Omron CX-Programmer project NewProject (CX-Programmer 9.74)

# PLC Transporte: CJ2M CPU31
I/O table (CPU CJ2M-CPU31): rack 0 slot 0 CJ1W-ID211; rack 0 slot 1 CJ1W-ID211; rack 0 slot 2 CJ1W-ID211; rack 0 slot 3 CJ1W-OD212; rack 0 slot 4 CJ1W-OD212; rack 0 slot 11 CJ2M-EIP21

## Data types
TYPE s_equip_ios : STRUCT  (* Equipamento - Entradas *)
  om : BOOL;  (* Ordem de marcha *)
  oma : BOOL;  (* Ordem de abrir *)
  omf : BOOL;  (* Ordem de fechar *)
  rm : BOOL;  (* Resposta de marcha *)
  fca : BOOL;  (* Fim de curso aberta *)
  fcf : BOOL;  (* Fim de curso fechada *)
  de : BOOL;  (* Defeito electrico *)
  pf_bmb : BOOL;  (* Pulsos de funcionamento da bomba *)
END_STRUCT END_TYPE
TYPE s_relogio : STRUCT  (* Dados de acerto e leitura de relógio *)
  pc_ano : INT;  (* Ano *)
  pc_mes : INT;  (* Mes *)
  pc_dia : INT;  (* Dia *)
  pc_dia_s : INT;  (* Dia da semana *)
  pc_hora : INT;  (* Hora *)
  pc_minuto : INT;  (* Minuto *)
  pc_segundo : INT;  (* Segundo *)
  rsv1 : INT Dimensions=[3];  (* RESERVA *)
  ano : INT;  (* Ano *)
  mes : INT;  (* Mes *)
  dia : INT;  (* Dia *)
  dia_s : INT;  (* Dia da semana *)
  hora : INT;  (* Hora *)
  minuto : INT;  (* Minuto *)
  segundo : INT;  (* Segundo *)
  rsv2 : INT Dimensions=[3];  (* RESERVA *)
END_STRUCT END_TYPE
TYPE s_caudal : STRUCT  (* Dados do caudalimetro *)
  tti : BOOL;  (* Impulso de totalização *)
  x0_1 : BOOL;  (* RESERVA *)
  x0_2 : BOOL;  (* RESERVA *)
  x0_3 : BOOL;  (* RESERVA *)
  fm : BOOL;  (* Falha de caudal *)
  rem : BOOL;  (* Totalizador local/remoto *)
  rem_ok : BOOL;  (* OK para ir buscar o valor do totalizador remoto *)
  inj_ini : BOOL;  (* Inicio da injecção *)
  x0_8 : BOOL;  (* RESERVA *)
  x0_9 : BOOL;  (* RESERVA *)
  x0_10 : BOOL;  (* RESERVA *)
  x0_11 : BOOL;  (* RESERVA *)
  x0_12 : BOOL;  (* RESERVA *)
  x0_13 : BOOL;  (* RESERVA *)
  x0_14 : BOOL;  (* RESERVA *)
  x0_15 : BOOL;  (* RESERVA *)
  prod : INT;  (* Produto *)
  rsv1 : INT Dimensions=[6];  (* RESERVA *)
  tti_x : REAL;  (* Valor do impulso *)
  tt_rem : REAL;  (* Totalizador remoto *)
  tt_rem_old : REAL;  (* Totalizador remoto antigo *)
  tt_inj : REAL;  (* Totalizador de injecção *)
  tt_p : REAL;  (* Totalizador parcial *)
  tt_g : REAL;  (* Totalizador global *)
END_STRUCT END_TYPE
TYPE s_deposito_p : STRUCT  (* Deposito de produto *)
  prod : INT;  (* Produto *)
  s_aut : BOOL;  (* Automatico *)
  mdp : BOOL;  (* Disponibilidade *)
  ndp : BOOL;  (* Não disponivel *)
  dgm : BOOL;  (* Defeito geral de maquina *)
  rst : BOOL;  (* Reset *)
  on : BOOL;  (* Deposito ligado *)
  oms_red : BOOL;  (* Lampada FLASH vermelho *)
  oms_green : BOOL;  (* Lampada FLASH verde *)
  rsv1 : INT Dimensions=[8];  (* Reserva *)
END_STRUCT END_TYPE
TYPE s_equip_bits : STRUCT  (* Equipamento - Bits auxiliares *)
  s_aut : BOOL;  (* Automatico *)
  mdp : BOOL;  (* Disponibilidade *)
  ndp : BOOL;  (* Não disponivel *)
  dgm : BOOL;  (* Defeito geral de maquina *)
  rst : BOOL;  (* Reset *)
  cfa : BOOL;  (* Condição de funcionamento automatico *)
  cfm : BOOL;  (* Condição de funcionamento manual *)
  cfaa : BOOL;  (* Condição de funcionamento automatico abrir *)
  cfaf : BOOL;  (* Condição de funcionamento automatico fechar *)
  cfma : BOOL;  (* Condição de funcionamento manual abrir *)
  cfmf : BOOL;  (* Condição de funcionamento manual fechar *)
  st_hmi : BOOL;  (* Arranque HMI *)
  sp_hmi : BOOL;  (* Paragem HMI *)
  p_hmi : BOOL;  (* Pausa HMI *)
END_STRUCT END_TYPE
TYPE s_equip_defs : STRUCT  (* Equipamentos - Defeitos *)
  fm : BOOL;  (* Falha de marcha *)
  fma : BOOL;  (* Falha de manobra abrir *)
  fmf : BOOL;  (* Falha de manobra fechar *)
  de : BOOL;  (* Defeito electrico *)
  dv : BOOL;  (* Deposito vazio *)
END_STRUCT END_TYPE
TYPE s_equip : STRUCT  (* Equipamento *)
  ios : s_equip_ios;  (* Entradas *)
  bits : s_equip_bits;  (* Bits *)
  defs : s_equip_defs;  (* Defeitos *)
  es : INT;  (* Estado *)
  tm_b : INT;  (* Tempo entre bombagens *)
  rsv1 : INT Dimensions=[5];  (* Reserva *)
END_STRUCT END_TYPE

## Global symbols (name address type ; comment)
Actv_M E0_25101 INT
H0.00 BOOL  ; CDTs Visible
Auto_Transport FIFO
Auto_Trspt_EN E0_25100.06 BOOL
Last_Rqst E0_25102 INT
Priority_Array E0_25000 INT[100]
Tapete1 fb_eq_motor
Tapete2 fb_eq_motor
Tapete3 fb_eq_motor
Tapete4 fb_eq_motor
Trspt_Array_Full E0_25100.07 BOOL
Trspt_Free E0_25100.14 BOOL
comm_M1_Rqst E0_25100.00 BOOL  ; From MES1
comm_M2_Rqst E0_25100.01 BOOL  ; From MES1
comm_M3_Rqst E0_25100.02 BOOL  ; From MES1
comm_M4_Rqst E0_25100.03 BOOL  ; From MES1
comm_M5_Rqst E0_25100.04 BOOL  ; From MES2
comm_M6_Rqst E0_25100.05 BOOL  ; From MES2
fb_eq_vc_M1 fb_eq_valvula
fb_eq_vc_M2 fb_eq_valvula
fb_eq_vc_M3 fb_eq_valvula
fb_eq_vc_M4 fb_eq_valvula
fb_eq_vc_M5 fb_eq_valvula
fb_eq_vc_M6 fb_eq_valvula
fb_eq_vd_M1 fb_eq_valvula
fb_eq_vd_M2 fb_eq_valvula
fb_eq_vd_M3 fb_eq_valvula
fb_eq_vd_M4 fb_eq_valvula
fb_eq_vd_M5 fb_eq_valvula
fb_eq_vd_M6 fb_eq_valvula

## Program Transporte (cyclic task 0)
Local symbols
Alarme_naa_t1 D0.01 BOOL
Alim_M1 W1.00 BOOL
Alim_M2 W1.01 BOOL
Alim_M3 W1.02 BOOL
Alim_M4 W1.03 BOOL
Alim_M5 W1.04 BOOL
Alim_M6 W1.05 BOOL
Carga_M1 D10050.05 BOOL  ; Ordem de alimentação da Máquina 1
Carga_M2 D10100.05 BOOL  ; Ordem de alimentação da Máquina 2
Carga_M3 D10150.05 BOOL  ; Ordem de alimentação da Máquina 3
Carga_M4 D10200.05 BOOL  ; Ordem de alimentação da Máquina 4
Carga_M5 D10250.05 BOOL  ; Ordem de alimentação da Máquina 5
Carga_M6 D10300.05 BOOL  ; Ordem de alimentação da Máquina 6
Encravamento_t2 W0.00 BOOL
M1_TrpRqst_Holder W2.02 BOOL
M2_TrpRqstHolder BOOL
M2_TrpRqst_Holder W2.00 BOOL
M3_TrpRqst_Holder W2.01 BOOL
M4_TrpRqst_Holder W2.03 BOOL
M5_TrpRqst_Holder W2.05 BOOL
M6_TrpRqst_Holder W2.04 BOOL
Tapete1 D10 STRUCT s_equip
Tapete2 D20 STRUCT s_equip
Tapete3 D30 STRUCT s_equip
Tapete4 D40 STRUCT s_equip
Transporte_M1 E0_25100.08 BOOL  ; Ordem de alimentação do Silo da Máquina 1
Transporte_M2 E0_25100.09 BOOL  ; Ordem de alimentação do Silo da Máquina 2
Transporte_M3 E0_25100.10 BOOL  ; Ordem de alimentação do Silo da Máquina 3
Transporte_M4 E0_25100.11 BOOL  ; Ordem de alimentação do Silo da Máquina 4
Transporte_M5 E0_25100.12 BOOL  ; Ordem de alimentação do Silo da Máquina 5
Transporte_M6 E0_25100.13 BOOL  ; Ordem de alimentação do Silo da Máquina 6
al_na_m1 D2.01 BOOL  ; Nivel alto estabilizado maquina 1
al_na_m2 D2.02 BOOL  ; Nivel alto estabilizado maquina 2
al_na_m3 D2.03 BOOL  ; Nivel alto estabilizado maquina 3
al_na_m4 D2.04 BOOL  ; Nivel alto estabilizado maquina 4
al_na_m5 D2.05 BOOL  ; Nivel alto estabilizado maquina 5
al_na_m6 D2.06 BOOL  ; Nivel alto estabilizado maquina 6
al_nb_m1 D1.01 BOOL  ; Nivel baixo estabilizado maquina 1
al_nb_m2 D1.02 BOOL  ; Nivel baixo estabilizado maquina 2
al_nb_m3 D1.03 BOOL  ; Nivel baixo estabilizado maquina 3
al_nb_m4 D1.04 BOOL  ; Nivel baixo estabilizado maquina 4
al_nb_m5 D1.05 BOOL  ; Nivel baixo estabilizado maquina 5
al_nb_m6 D1.06 BOOL  ; Nivel baixo estabilizado maquina 6
cmd_rst_vc_M1 D10050.03 BOOL  ; Comando de reset da Razeira da Máquina 1
cmd_rst_vc_M2 D10100.03 BOOL  ; Comando de reset da Razeira da Máquina 2
cmd_rst_vc_M3 D10150.03 BOOL  ; Comando de reset da Razeira da Máquina 3
cmd_rst_vc_M4 D10200.03 BOOL  ; Comando de reset da Razeira da Máquina 4
cmd_rst_vc_M5 D10250.03 BOOL  ; Comando de reset da Razeira da Máquina 5
cmd_rst_vc_M6 D10300.03 BOOL  ; Comando de reset da Razeira da Máquina 6
cmd_tp3_M1 D10050.06 BOOL  ; Ordem de marcha Tapete 3 a partir da Máquina 1
cmd_tp3_M2 D10100.06 BOOL  ; Ordem de marcha Tapete 3 a partir da Máquina 2
cmd_tp3_M3 D10150.06 BOOL  ; Ordem de marcha Tapete 3 a partir da Máquina 3
cmd_tp3_M4 D10200.06 BOOL  ; Ordem de marcha Tapete 3 a partir da Máquina 4
cmd_tp3_M5 D10250.06 BOOL  ; Ordem de marcha Tapete 3 a partir da Máquina 5
cmd_tp3_M6 D10300.06 BOOL  ; Ordem de marcha Tapete 3 a partir da Máquina 6
cmd_tp4_M1 D10050.07 BOOL  ; Ordem de marcha Tapete 4 a partir da Máquina 1
cmd_tp4_M2 D10100.07 BOOL  ; Ordem de marcha Tapete 4 a partir da Máquina 2
cmd_tp4_M3 D10150.07 BOOL  ; Ordem de marcha Tapete 4 a partir da Máquina 3
cmd_tp4_M4 D10200.07 BOOL  ; Ordem de marcha Tapete 4 a partir da Máquina 4
cmd_tp4_M5 D10250.07 BOOL  ; Ordem de marcha Tapete 4 a partir da Máquina 5
cmd_tp4_M6 D10300.07 BOOL  ; Ordem de marcha Tapete 4 a partir da Máquina 6
de_t1 1.00 BOOL  ; Disparo termico no tapete 1
de_t2 1.01 BOOL  ; Disparo termico no tapete 2
de_t3 1.02 BOOL  ; Disparo termico no tapete 3
de_t4 1.03 BOOL  ; Disparo termico no tapete 4
disp_transporte D0.03 BOOL
fca_vd_m1 2.00 BOOL  ; Valvula desviadora aberta - maquina 1
fca_vd_m2 2.02 BOOL  ; Valvula desviadora aberta - maquina 2
fca_vd_m3 2.04 BOOL  ; Valvula desviadora aberta - maquina 3
fca_vd_m4 2.06 BOOL  ; Valvula desviadora aberta - maquina 4
fca_vd_m5 2.08 BOOL  ; Valvula desviadora aberta - maquina 5
fca_vd_m6 2.10 BOOL  ; Valvula desviadora aberta - maquina 6
fcf_vc_m1 1.04 BOOL  ; Razeira de carga fechada - maquina 1
fcf_vc_m2 1.05 BOOL  ; Razeira de carga fechada - maquina 2
fcf_vc_m3 1.06 BOOL  ; Razeira de carga fechada - maquina 3
fcf_vc_m4 1.07 BOOL  ; Razeira de carga fechada - maquina 4
fcf_vc_m5 1.08 BOOL  ; Razeira de carga fechada - maquina 5
fcf_vc_m6 1.09 BOOL  ; Razeira de carga fechada - maquina 6
fcf_vd_m1 2.01 BOOL  ; Valvula desviadora fechada - maquina 1
fcf_vd_m2 2.03 BOOL  ; Valvula desviadora fechada - maquina 2
fcf_vd_m3 2.05 BOOL  ; Valvula desviadora fechada - maquina 3
fcf_vd_m4 2.07 BOOL  ; Valvula desviadora fechada - maquina 4
fcf_vd_m5 2.09 BOOL  ; Valvula desviadora fechada - maquina 5
fcf_vd_m6 2.11 BOOL  ; Valvula desviadora fechada - maquina 6
msb_1 BOOL
na_m1 0.02 BOOL  ; Nivel alto na moega de carga maquina 1
na_m2 0.04 BOOL  ; Nivel alto na moega de carga maquina 2
na_m3 0.06 BOOL  ; Nivel alto na moega de carga maquina 3
na_m4 0.08 BOOL  ; Nivel alto na moega de carga maquina 4
na_m5 0.10 BOOL  ; Nivel alto na moega de carga maquina 5
na_m6 0.12 BOOL  ; Nivel alto na moega de carga maquina 6
naa_t1 0.14 BOOL  ; Nivel muito alto no tapete 1
naa_t1_tp D0.00 BOOL
nb_m1 0.03 BOOL  ; Nivel baixo na moega de carga maquina 1
nb_m2 0.05 BOOL  ; Nivel baixo na moega de carga maquina 2
nb_m3 0.07 BOOL  ; Nivel baixo na moega de carga maquina 3
nb_m4 0.09 BOOL  ; Nivel baixo na moega de carga maquina 4
nb_m5 0.11 BOOL  ; Nivel baixo na moega de carga maquina 5
nb_m6 0.13 BOOL  ; Nivel baixo na moega de carga maquina 6
om_t1 3.00 BOOL  ; Ordem de marcha tapete 1
om_t2 3.01 BOOL  ; Ordem de marcha tapete 2
om_t3 3.02 BOOL  ; Ordem de marcha tapete 3
om_t4 3.03 BOOL  ; Ordem de marcha tapete 4
oma_vc_m1 3.04 BOOL  ; Abrir razeira de carga - maquina 1
oma_vc_m2 3.06 BOOL  ; Abrir razeira de carga - maquina 2
oma_vc_m3 3.08 BOOL  ; Abrir razeira de carga - maquina 3
oma_vc_m4 3.10 BOOL  ; Abrir razeira de carga - maquina 4
oma_vc_m5 3.12 BOOL  ; Abrir razeira de carga - maquina 5
oma_vc_m6 3.14 BOOL  ; Abrir razeira de carga - maquina 6
oma_vd_m1 4.01 BOOL  ; Abrir valvula desviadora - maquina 1
oma_vd_m2 4.03 BOOL  ; Abrir valvula desviadora - maquina 2
oma_vd_m3 4.05 BOOL  ; Abrir valvula desviadora - maquina 3
oma_vd_m4 4.07 BOOL  ; Abrir valvula desviadora - maquina 4
oma_vd_m5 4.09 BOOL  ; Abrir valvula desviadora - maquina 5
oma_vd_m6 4.11 BOOL  ; Abrir valvula desviadora - maquina 6
omf_vc_m1 3.05 BOOL  ; Fechar razeira de carga - maquina 1
omf_vc_m2 3.07 BOOL  ; Fechar razeira de carga - maquina 2
omf_vc_m3 3.09 BOOL  ; Fechar razeira de carga - maquina 3
omf_vc_m4 3.11 BOOL  ; Fechar razeira de carga - maquina 4
omf_vc_m5 3.13 BOOL  ; Fechar razeira de carga - maquina 5
omf_vc_m6 3.15 BOOL  ; Fechar razeira de carga - maquina 6
omf_vd_m1 4.00 BOOL  ; Fechar valvula desviadora - maquina 1
omf_vd_m2 4.02 BOOL  ; Fechar valvula desviadora - maquina 2
omf_vd_m3 4.04 BOOL  ; Fechar valvula desviadora - maquina 3
omf_vd_m4 4.06 BOOL  ; Fechar valvula desviadora - maquina 4
omf_vd_m5 4.08 BOOL  ; Fechar valvula desviadora - maquina 5
omf_vd_m6 4.10 BOOL  ; Fechar valvula desviadora - maquina 6
pe_transporte 0.00 BOOL  ; Botoneira de Emergência
rem_transporte 0.01 BOOL  ; Automatico
rm_t1 1.10 BOOL  ; Resposta de marcha tapete 1
rm_t2 1.11 BOOL  ; Resposta de marcha tapete 2
rm_t3 1.12 BOOL  ; Resposta de marcha tapete 3
rm_t4 1.13 BOOL  ; Resposta de marcha tapete 4
rm_transporte D0.05 BOOL
so_1alim D0.02 BOOL
stop_transporte D0.04 BOOL
vc_M1 D100 STRUCT s_equip
vc_M2 D110 STRUCT s_equip
vc_M3 D120 STRUCT s_equip
vc_M4 D130 STRUCT s_equip
vc_M5 D140 STRUCT s_equip
vc_M6 D150 STRUCT s_equip
vd_M1 D200 STRUCT s_equip
vd_M2 D210 STRUCT s_equip
vd_M3 D220 STRUCT s_equip
vd_M4 D230 STRUCT s_equip
vd_M5 D240 STRUCT s_equip
vd_M6 D250 STRUCT s_equip

### Section Valvulas

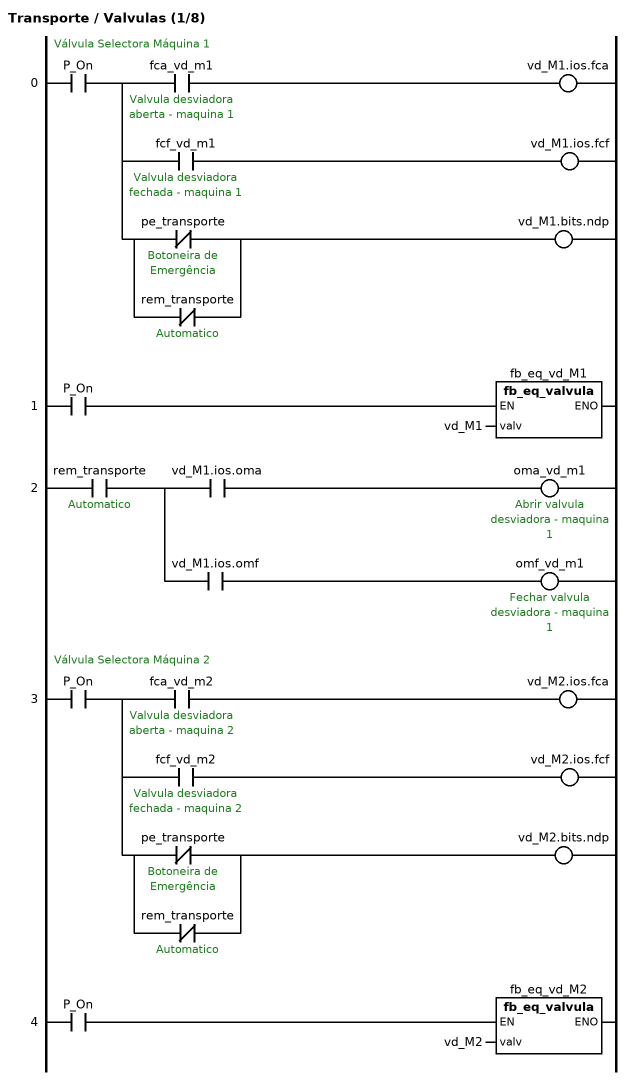
; rung 0: Válvula Selectora Máquina 1
LD P_On
OUT TR0
AND fca_vd_m1  ; Valvula desviadora aberta - maquina 1
OUT vd_M1.ios.fca
LD TR0
AND fcf_vd_m1  ; Valvula desviadora fechada - maquina 1
OUT vd_M1.ios.fcf
LD TR0
LDNOT pe_transporte  ; Botoneira de Emergência
ORNOT rem_transporte  ; Automatico
ANDLD
OUT vd_M1.bits.ndp
; rung 1
LD P_On
CALL fb_eq_vd_M1 : fb_eq_valvula (valv := vd_M1)
; rung 2
LD rem_transporte  ; Automatico
OUT TR0
AND vd_M1.ios.oma
OUT oma_vd_m1  ; Abrir valvula desviadora - maquina 1
LD TR0
AND vd_M1.ios.omf
OUT omf_vd_m1  ; Fechar valvula desviadora - maquina 1
; rung 3: Válvula Selectora Máquina 2
LD P_On
OUT TR0
AND fca_vd_m2  ; Valvula desviadora aberta - maquina 2
OUT vd_M2.ios.fca
LD TR0
AND fcf_vd_m2  ; Valvula desviadora fechada - maquina 2
OUT vd_M2.ios.fcf
LD TR0
LDNOT pe_transporte  ; Botoneira de Emergência
ORNOT rem_transporte  ; Automatico
ANDLD
OUT vd_M2.bits.ndp
; rung 4
LD P_On
CALL fb_eq_vd_M2 : fb_eq_valvula (valv := vd_M2)

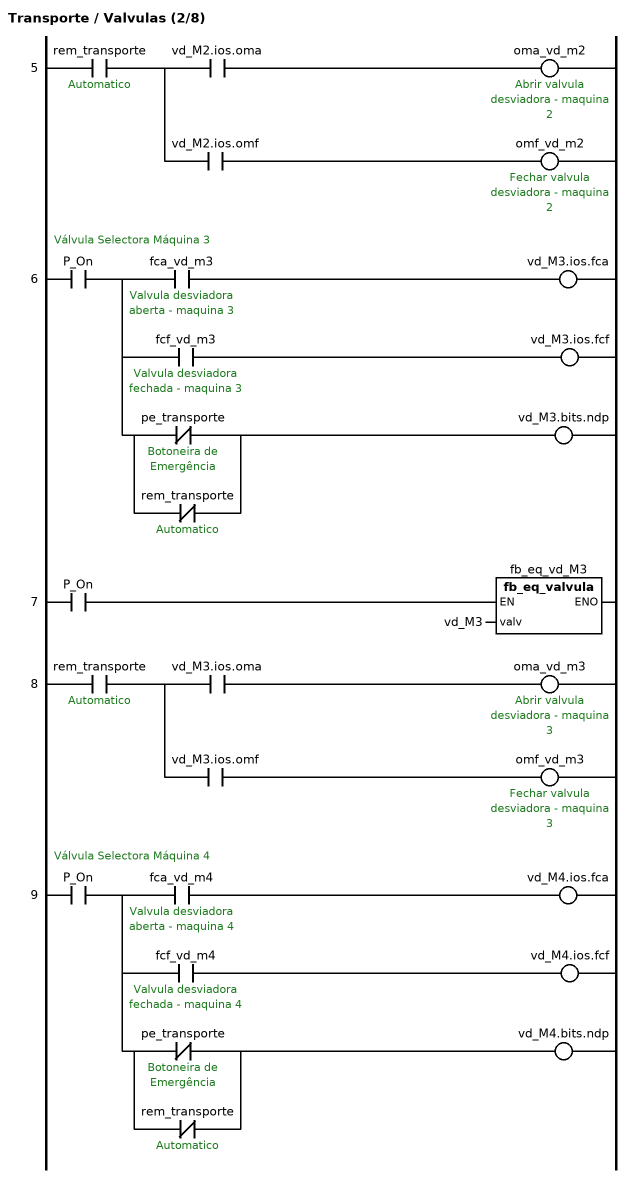
; rung 5
LD rem_transporte  ; Automatico
OUT TR0
AND vd_M2.ios.oma
OUT oma_vd_m2  ; Abrir valvula desviadora - maquina 2
LD TR0
AND vd_M2.ios.omf
OUT omf_vd_m2  ; Fechar valvula desviadora - maquina 2
; rung 6: Válvula Selectora Máquina 3
LD P_On
OUT TR0
AND fca_vd_m3  ; Valvula desviadora aberta - maquina 3
OUT vd_M3.ios.fca
LD TR0
AND fcf_vd_m3  ; Valvula desviadora fechada - maquina 3
OUT vd_M3.ios.fcf
LD TR0
LDNOT pe_transporte  ; Botoneira de Emergência
ORNOT rem_transporte  ; Automatico
ANDLD
OUT vd_M3.bits.ndp
; rung 7
LD P_On
CALL fb_eq_vd_M3 : fb_eq_valvula (valv := vd_M3)
; rung 8
LD rem_transporte  ; Automatico
OUT TR0
AND vd_M3.ios.oma
OUT oma_vd_m3  ; Abrir valvula desviadora - maquina 3
LD TR0
AND vd_M3.ios.omf
OUT omf_vd_m3  ; Fechar valvula desviadora - maquina 3
; rung 9: Válvula Selectora Máquina 4
LD P_On
OUT TR0
AND fca_vd_m4  ; Valvula desviadora aberta - maquina 4
OUT vd_M4.ios.fca
LD TR0
AND fcf_vd_m4  ; Valvula desviadora fechada - maquina 4
OUT vd_M4.ios.fcf
LD TR0
LDNOT pe_transporte  ; Botoneira de Emergência
ORNOT rem_transporte  ; Automatico
ANDLD
OUT vd_M4.bits.ndp

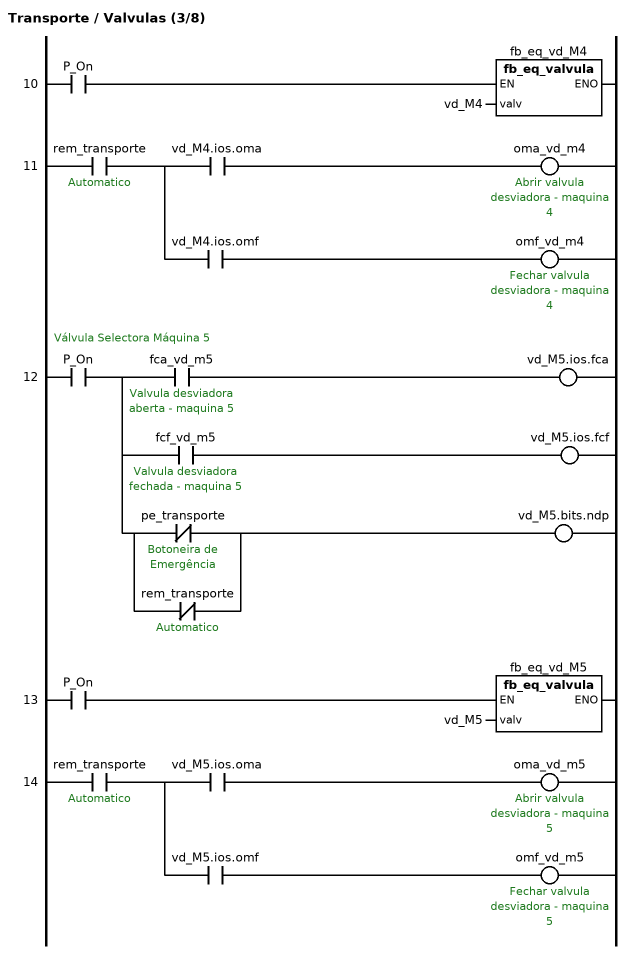
; rung 10
LD P_On
CALL fb_eq_vd_M4 : fb_eq_valvula (valv := vd_M4)
; rung 11
LD rem_transporte  ; Automatico
OUT TR0
AND vd_M4.ios.oma
OUT oma_vd_m4  ; Abrir valvula desviadora - maquina 4
LD TR0
AND vd_M4.ios.omf
OUT omf_vd_m4  ; Fechar valvula desviadora - maquina 4
; rung 12: Válvula Selectora Máquina 5
LD P_On
OUT TR0
AND fca_vd_m5  ; Valvula desviadora aberta - maquina 5
OUT vd_M5.ios.fca
LD TR0
AND fcf_vd_m5  ; Valvula desviadora fechada - maquina 5
OUT vd_M5.ios.fcf
LD TR0
LDNOT pe_transporte  ; Botoneira de Emergência
ORNOT rem_transporte  ; Automatico
ANDLD
OUT vd_M5.bits.ndp
; rung 13
LD P_On
CALL fb_eq_vd_M5 : fb_eq_valvula (valv := vd_M5)
; rung 14
LD rem_transporte  ; Automatico
OUT TR0
AND vd_M5.ios.oma
OUT oma_vd_m5  ; Abrir valvula desviadora - maquina 5
LD TR0
AND vd_M5.ios.omf
OUT omf_vd_m5  ; Fechar valvula desviadora - maquina 5

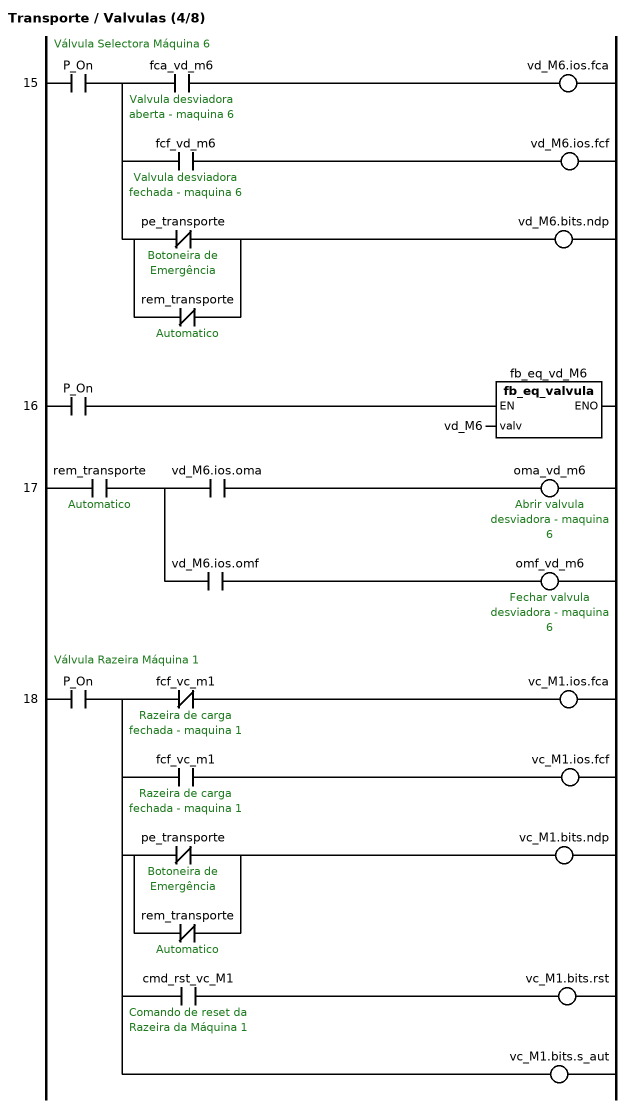
; rung 15: Válvula Selectora Máquina 6
LD P_On
OUT TR0
AND fca_vd_m6  ; Valvula desviadora aberta - maquina 6
OUT vd_M6.ios.fca
LD TR0
AND fcf_vd_m6  ; Valvula desviadora fechada - maquina 6
OUT vd_M6.ios.fcf
LD TR0
LDNOT pe_transporte  ; Botoneira de Emergência
ORNOT rem_transporte  ; Automatico
ANDLD
OUT vd_M6.bits.ndp
; rung 16
LD P_On
CALL fb_eq_vd_M6 : fb_eq_valvula (valv := vd_M6)
; rung 17
LD rem_transporte  ; Automatico
OUT TR0
AND vd_M6.ios.oma
OUT oma_vd_m6  ; Abrir valvula desviadora - maquina 6
LD TR0
AND vd_M6.ios.omf
OUT omf_vd_m6  ; Fechar valvula desviadora - maquina 6
; rung 18: Válvula Razeira Máquina 1
LD P_On
OUT TR0
ANDNOT fcf_vc_m1  ; Razeira de carga fechada - maquina 1
OUT vc_M1.ios.fca
LD TR0
AND fcf_vc_m1  ; Razeira de carga fechada - maquina 1
OUT vc_M1.ios.fcf
LD TR0
LDNOT pe_transporte  ; Botoneira de Emergência
ORNOT rem_transporte  ; Automatico
ANDLD
OUT vc_M1.bits.ndp
LD TR0
AND cmd_rst_vc_M1  ; Comando de reset da Razeira da Máquina 1
OUT vc_M1.bits.rst
LD TR0
OUT vc_M1.bits.s_aut

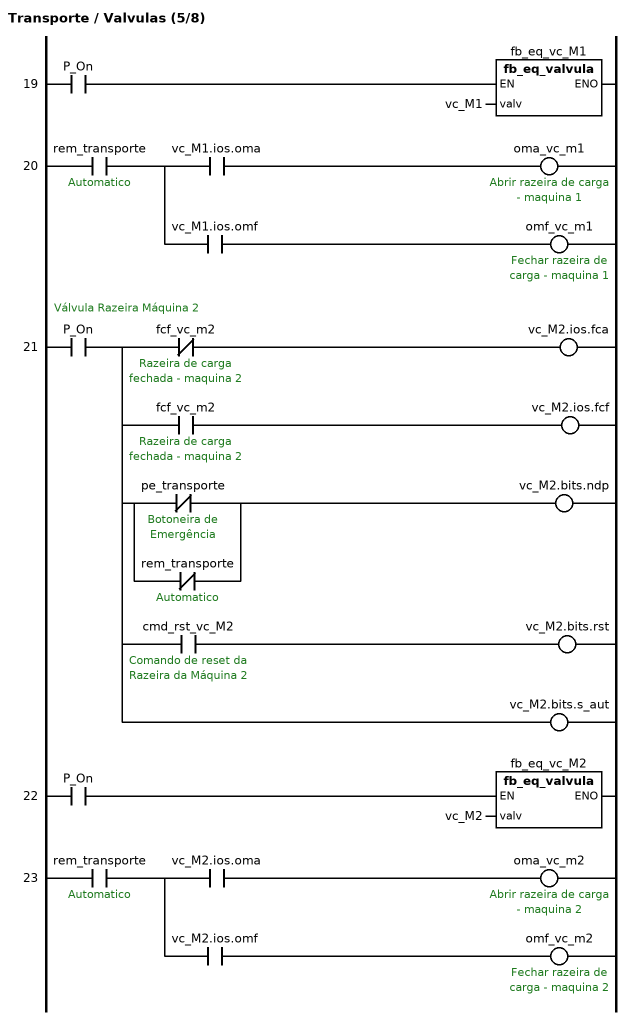
; rung 19
LD P_On
CALL fb_eq_vc_M1 : fb_eq_valvula (valv := vc_M1)
; rung 20
LD rem_transporte  ; Automatico
OUT TR0
AND vc_M1.ios.oma
OUT oma_vc_m1  ; Abrir razeira de carga - maquina 1
LD TR0
AND vc_M1.ios.omf
OUT omf_vc_m1  ; Fechar razeira de carga - maquina 1
; rung 21: Válvula Razeira Máquina 2
LD P_On
OUT TR0
ANDNOT fcf_vc_m2  ; Razeira de carga fechada - maquina 2
OUT vc_M2.ios.fca
LD TR0
AND fcf_vc_m2  ; Razeira de carga fechada - maquina 2
OUT vc_M2.ios.fcf
LD TR0
LDNOT pe_transporte  ; Botoneira de Emergência
ORNOT rem_transporte  ; Automatico
ANDLD
OUT vc_M2.bits.ndp
LD TR0
AND cmd_rst_vc_M2  ; Comando de reset da Razeira da Máquina 2
OUT vc_M2.bits.rst
LD TR0
OUT vc_M2.bits.s_aut
; rung 22
LD P_On
CALL fb_eq_vc_M2 : fb_eq_valvula (valv := vc_M2)
; rung 23
LD rem_transporte  ; Automatico
OUT TR0
AND vc_M2.ios.oma
OUT oma_vc_m2  ; Abrir razeira de carga - maquina 2
LD TR0
AND vc_M2.ios.omf
OUT omf_vc_m2  ; Fechar razeira de carga - maquina 2

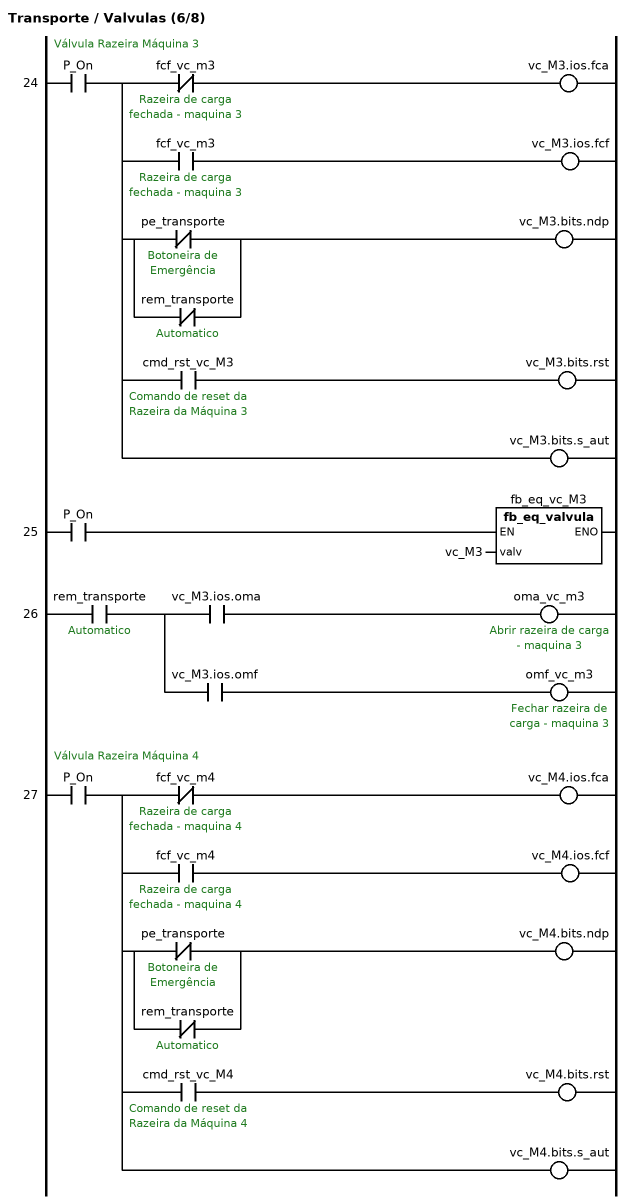
; rung 24: Válvula Razeira Máquina 3
LD P_On
OUT TR0
ANDNOT fcf_vc_m3  ; Razeira de carga fechada - maquina 3
OUT vc_M3.ios.fca
LD TR0
AND fcf_vc_m3  ; Razeira de carga fechada - maquina 3
OUT vc_M3.ios.fcf
LD TR0
LDNOT pe_transporte  ; Botoneira de Emergência
ORNOT rem_transporte  ; Automatico
ANDLD
OUT vc_M3.bits.ndp
LD TR0
AND cmd_rst_vc_M3  ; Comando de reset da Razeira da Máquina 3
OUT vc_M3.bits.rst
LD TR0
OUT vc_M3.bits.s_aut
; rung 25
LD P_On
CALL fb_eq_vc_M3 : fb_eq_valvula (valv := vc_M3)
; rung 26
LD rem_transporte  ; Automatico
OUT TR0
AND vc_M3.ios.oma
OUT oma_vc_m3  ; Abrir razeira de carga - maquina 3
LD TR0
AND vc_M3.ios.omf
OUT omf_vc_m3  ; Fechar razeira de carga - maquina 3
; rung 27: Válvula Razeira Máquina 4
LD P_On
OUT TR0
ANDNOT fcf_vc_m4  ; Razeira de carga fechada - maquina 4
OUT vc_M4.ios.fca
LD TR0
AND fcf_vc_m4  ; Razeira de carga fechada - maquina 4
OUT vc_M4.ios.fcf
LD TR0
LDNOT pe_transporte  ; Botoneira de Emergência
ORNOT rem_transporte  ; Automatico
ANDLD
OUT vc_M4.bits.ndp
LD TR0
AND cmd_rst_vc_M4  ; Comando de reset da Razeira da Máquina 4
OUT vc_M4.bits.rst
LD TR0
OUT vc_M4.bits.s_aut

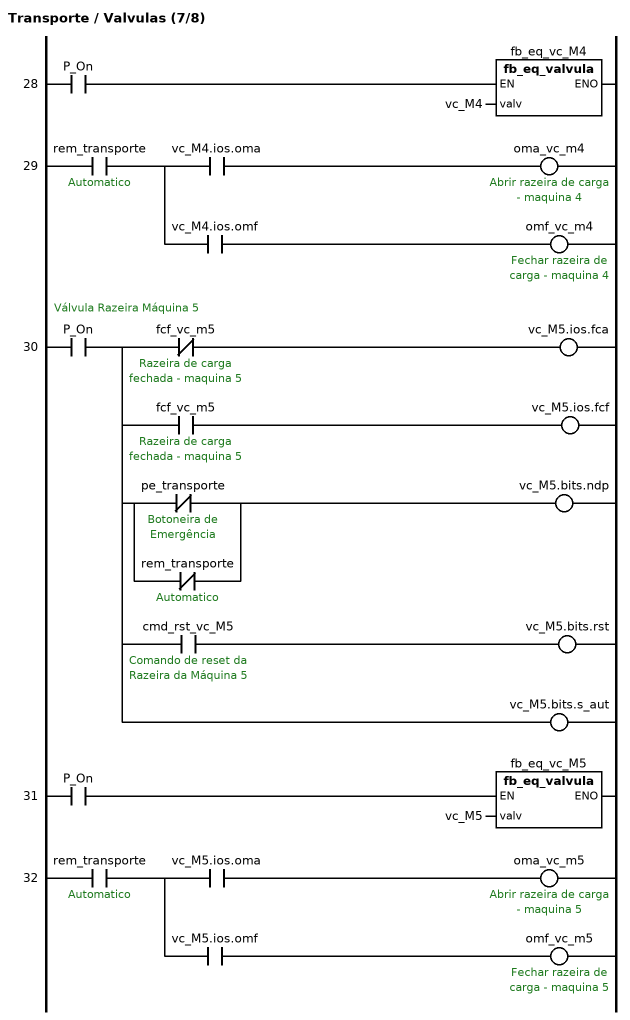
; rung 28
LD P_On
CALL fb_eq_vc_M4 : fb_eq_valvula (valv := vc_M4)
; rung 29
LD rem_transporte  ; Automatico
OUT TR0
AND vc_M4.ios.oma
OUT oma_vc_m4  ; Abrir razeira de carga - maquina 4
LD TR0
AND vc_M4.ios.omf
OUT omf_vc_m4  ; Fechar razeira de carga - maquina 4
; rung 30: Válvula Razeira Máquina 5
LD P_On
OUT TR0
ANDNOT fcf_vc_m5  ; Razeira de carga fechada - maquina 5
OUT vc_M5.ios.fca
LD TR0
AND fcf_vc_m5  ; Razeira de carga fechada - maquina 5
OUT vc_M5.ios.fcf
LD TR0
LDNOT pe_transporte  ; Botoneira de Emergência
ORNOT rem_transporte  ; Automatico
ANDLD
OUT vc_M5.bits.ndp
LD TR0
AND cmd_rst_vc_M5  ; Comando de reset da Razeira da Máquina 5
OUT vc_M5.bits.rst
LD TR0
OUT vc_M5.bits.s_aut
; rung 31
LD P_On
CALL fb_eq_vc_M5 : fb_eq_valvula (valv := vc_M5)
; rung 32
LD rem_transporte  ; Automatico
OUT TR0
AND vc_M5.ios.oma
OUT oma_vc_m5  ; Abrir razeira de carga - maquina 5
LD TR0
AND vc_M5.ios.omf
OUT omf_vc_m5  ; Fechar razeira de carga - maquina 5

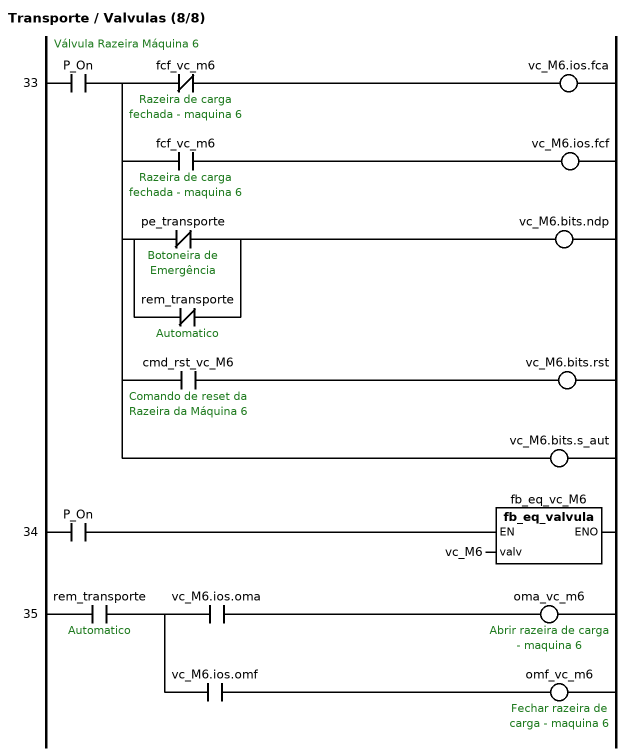
; rung 33: Válvula Razeira Máquina 6
LD P_On
OUT TR0
ANDNOT fcf_vc_m6  ; Razeira de carga fechada - maquina 6
OUT vc_M6.ios.fca
LD TR0
AND fcf_vc_m6  ; Razeira de carga fechada - maquina 6
OUT vc_M6.ios.fcf
LD TR0
LDNOT pe_transporte  ; Botoneira de Emergência
ORNOT rem_transporte  ; Automatico
ANDLD
OUT vc_M6.bits.ndp
LD TR0
AND cmd_rst_vc_M6  ; Comando de reset da Razeira da Máquina 6
OUT vc_M6.bits.rst
LD TR0
OUT vc_M6.bits.s_aut
; rung 34
LD P_On
CALL fb_eq_vc_M6 : fb_eq_valvula (valv := vc_M6)
; rung 35
LD rem_transporte  ; Automatico
OUT TR0
AND vc_M6.ios.oma
OUT oma_vc_m6  ; Abrir razeira de carga - maquina 6
LD TR0
AND vc_M6.ios.omf
OUT omf_vc_m6  ; Fechar razeira de carga - maquina 6

### Section Tapetes

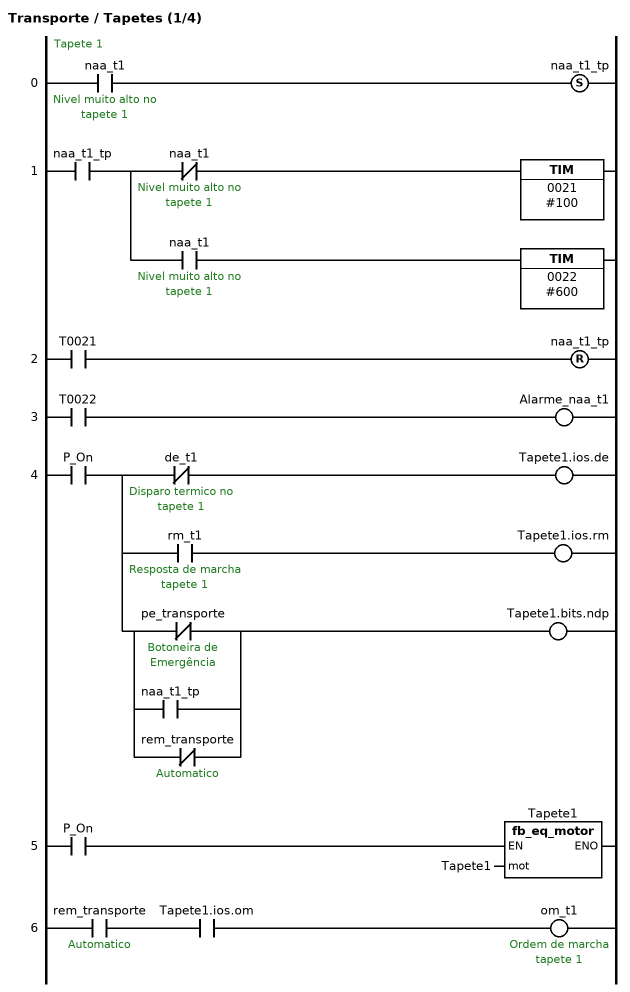
; rung 0: Tapete 1
LD naa_t1  ; Nivel muito alto no tapete 1
SET naa_t1_tp
; rung 1
LD naa_t1_tp
OUT TR0
ANDNOT naa_t1  ; Nivel muito alto no tapete 1
TIM 0021 #100
LD TR0
AND naa_t1  ; Nivel muito alto no tapete 1
TIM 0022 #600
; rung 2
LD T0021
RSET naa_t1_tp
; rung 3
LD T0022
OUT Alarme_naa_t1
; rung 4
LD P_On
OUT TR0
ANDNOT de_t1  ; Disparo termico no tapete 1
OUT Tapete1.ios.de
LD TR0
AND rm_t1  ; Resposta de marcha tapete 1
OUT Tapete1.ios.rm
LD TR0
LDNOT pe_transporte  ; Botoneira de Emergência
OR naa_t1_tp
ORNOT rem_transporte  ; Automatico
ANDLD
OUT Tapete1.bits.ndp
; rung 5
LD P_On
CALL Tapete1 : fb_eq_motor (mot := Tapete1)
; rung 6
LD rem_transporte  ; Automatico
AND Tapete1.ios.om
OUT om_t1  ; Ordem de marcha tapete 1

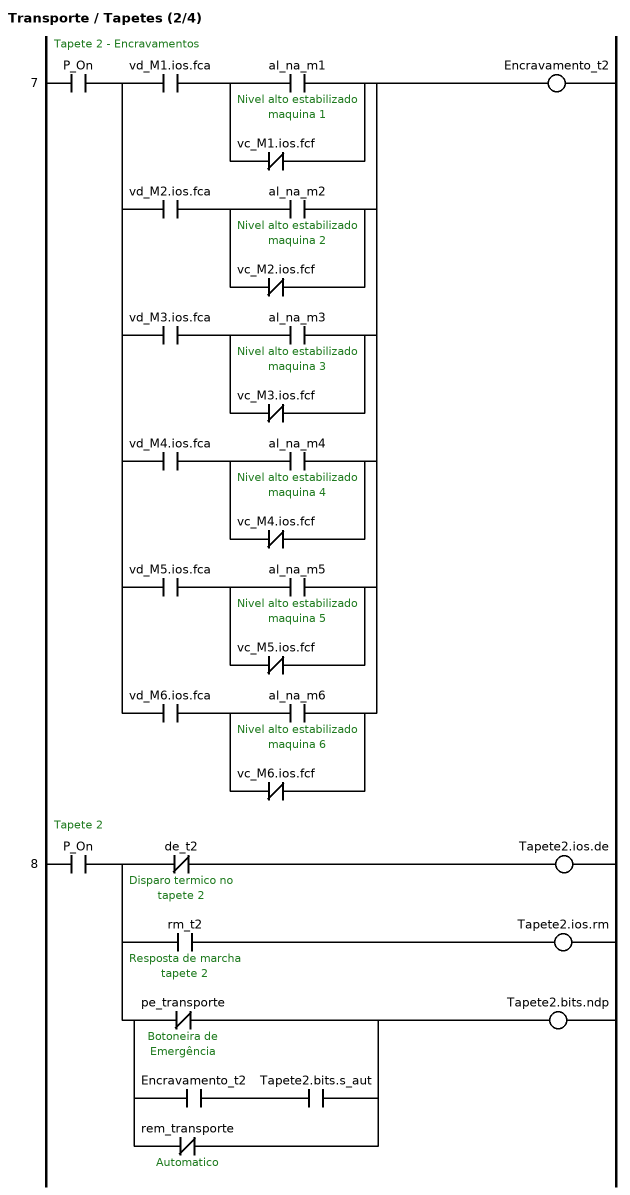
; rung 7: Tapete 2 - Encravamentos
LD P_On
LD vd_M1.ios.fca
LD al_na_m1  ; Nivel alto estabilizado maquina 1
ORNOT vc_M1.ios.fcf
ANDLD
LD vd_M2.ios.fca
LD al_na_m2  ; Nivel alto estabilizado maquina 2
ORNOT vc_M2.ios.fcf
ANDLD
ORLD
LD vd_M3.ios.fca
LD al_na_m3  ; Nivel alto estabilizado maquina 3
ORNOT vc_M3.ios.fcf
ANDLD
ORLD
LD vd_M4.ios.fca
LD al_na_m4  ; Nivel alto estabilizado maquina 4
ORNOT vc_M4.ios.fcf
ANDLD
ORLD
LD vd_M5.ios.fca
LD al_na_m5  ; Nivel alto estabilizado maquina 5
ORNOT vc_M5.ios.fcf
ANDLD
ORLD
LD vd_M6.ios.fca
LD al_na_m6  ; Nivel alto estabilizado maquina 6
ORNOT vc_M6.ios.fcf
ANDLD
ORLD
ANDLD
OUT Encravamento_t2
; rung 8: Tapete 2
LD P_On
OUT TR0
ANDNOT de_t2  ; Disparo termico no tapete 2
OUT Tapete2.ios.de
LD TR0
AND rm_t2  ; Resposta de marcha tapete 2
OUT Tapete2.ios.rm
LD TR0
LDNOT pe_transporte  ; Botoneira de Emergência
LD Encravamento_t2
AND Tapete2.bits.s_aut
ORLD
ORNOT rem_transporte  ; Automatico
ANDLD
OUT Tapete2.bits.ndp

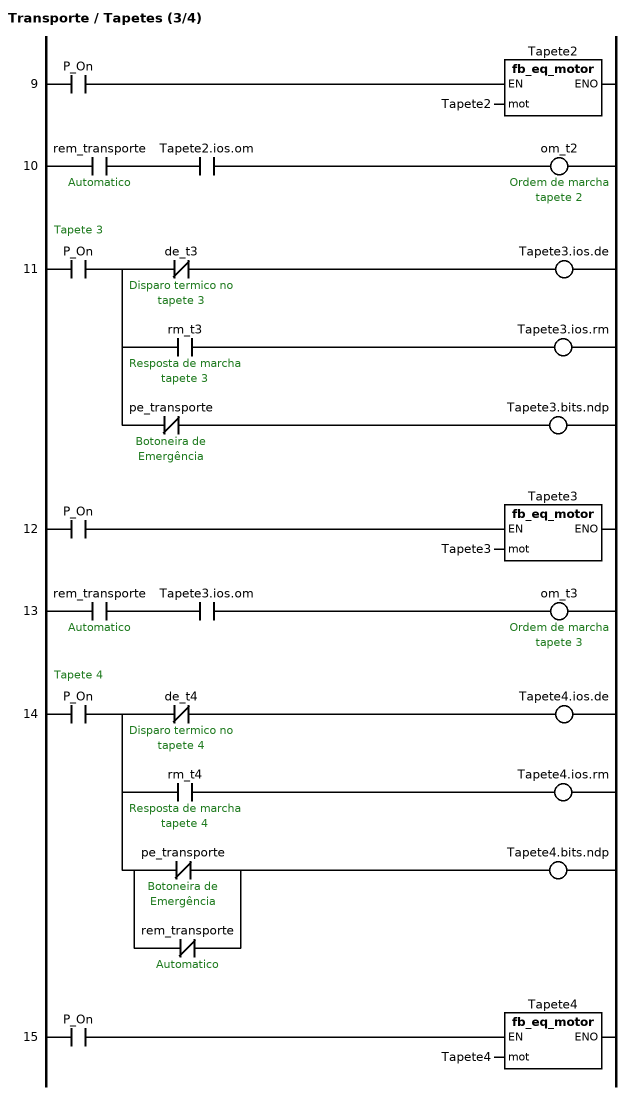
; rung 9
LD P_On
CALL Tapete2 : fb_eq_motor (mot := Tapete2)
; rung 10
LD rem_transporte  ; Automatico
AND Tapete2.ios.om
OUT om_t2  ; Ordem de marcha tapete 2
; rung 11: Tapete 3
LD P_On
OUT TR0
ANDNOT de_t3  ; Disparo termico no tapete 3
OUT Tapete3.ios.de
LD TR0
AND rm_t3  ; Resposta de marcha tapete 3
OUT Tapete3.ios.rm
LD TR0
ANDNOT pe_transporte  ; Botoneira de Emergência
OUT Tapete3.bits.ndp
; rung 12
LD P_On
CALL Tapete3 : fb_eq_motor (mot := Tapete3)
; rung 13
LD rem_transporte  ; Automatico
AND Tapete3.ios.om
OUT om_t3  ; Ordem de marcha tapete 3
; rung 14: Tapete 4
LD P_On
OUT TR0
ANDNOT de_t4  ; Disparo termico no tapete 4
OUT Tapete4.ios.de
LD TR0
AND rm_t4  ; Resposta de marcha tapete 4
OUT Tapete4.ios.rm
LD TR0
LDNOT pe_transporte  ; Botoneira de Emergência
ORNOT rem_transporte  ; Automatico
ANDLD
OUT Tapete4.bits.ndp
; rung 15
LD P_On
CALL Tapete4 : fb_eq_motor (mot := Tapete4)

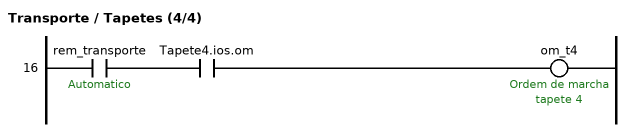
; rung 16
LD rem_transporte  ; Automatico
AND Tapete4.ios.om
OUT om_t4  ; Ordem de marcha tapete 4

### Section CFM_Tapetes

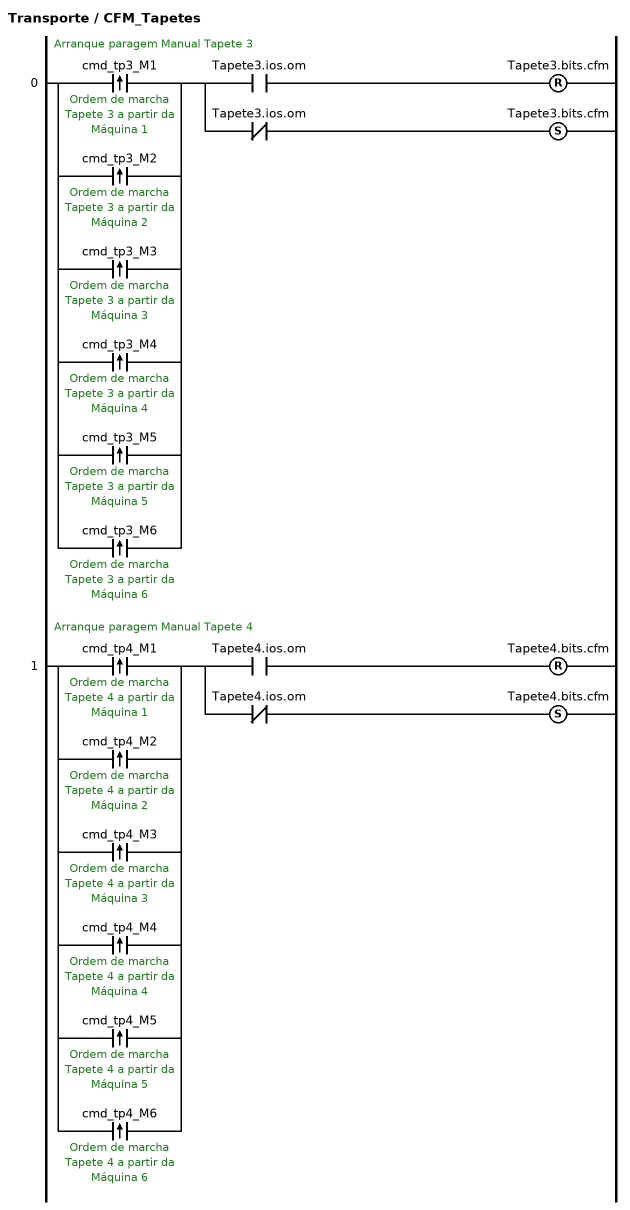
; rung 0: Arranque paragem Manual Tapete 3
@LD cmd_tp3_M1  ; Ordem de marcha Tapete 3 a partir da Máquina 1
@OR cmd_tp3_M2  ; Ordem de marcha Tapete 3 a partir da Máquina 2
@OR cmd_tp3_M3  ; Ordem de marcha Tapete 3 a partir da Máquina 3
@OR cmd_tp3_M4  ; Ordem de marcha Tapete 3 a partir da Máquina 4
@OR cmd_tp3_M5  ; Ordem de marcha Tapete 3 a partir da Máquina 5
@OR cmd_tp3_M6  ; Ordem de marcha Tapete 3 a partir da Máquina 6
OUT TR0
AND Tapete3.ios.om
RSET Tapete3.bits.cfm
LD TR0
ANDNOT Tapete3.ios.om
SET Tapete3.bits.cfm
; rung 1: Arranque paragem Manual Tapete 4
@LD cmd_tp4_M1  ; Ordem de marcha Tapete 4 a partir da Máquina 1
@OR cmd_tp4_M2  ; Ordem de marcha Tapete 4 a partir da Máquina 2
@OR cmd_tp4_M3  ; Ordem de marcha Tapete 4 a partir da Máquina 3
@OR cmd_tp4_M4  ; Ordem de marcha Tapete 4 a partir da Máquina 4
@OR cmd_tp4_M5  ; Ordem de marcha Tapete 4 a partir da Máquina 5
@OR cmd_tp4_M6  ; Ordem de marcha Tapete 4 a partir da Máquina 6
OUT TR0
AND Tapete4.ios.om
RSET Tapete4.bits.cfm
LD TR0
ANDNOT Tapete4.ios.om
SET Tapete4.bits.cfm

### Section CFA

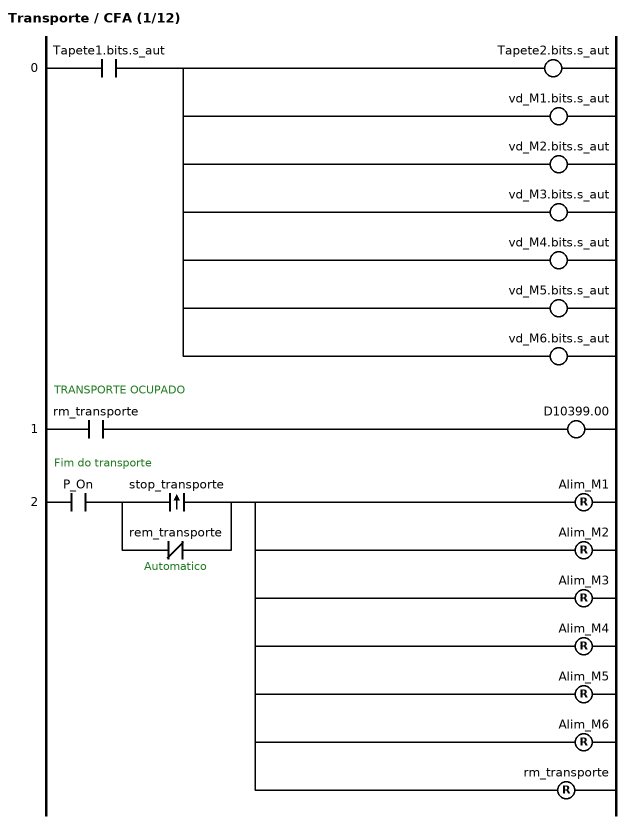
; rung 0
LD Tapete1.bits.s_aut
OUT Tapete2.bits.s_aut
OUT vd_M1.bits.s_aut
OUT vd_M2.bits.s_aut
OUT vd_M3.bits.s_aut
OUT vd_M4.bits.s_aut
OUT vd_M5.bits.s_aut
OUT vd_M6.bits.s_aut
; rung 1: TRANSPORTE OCUPADO
LD rm_transporte
OUT D10399.00
; rung 2: Fim do transporte
LD P_On
@LD stop_transporte
ORNOT rem_transporte  ; Automatico
ANDLD
RSET Alim_M1
RSET Alim_M2
RSET Alim_M3
RSET Alim_M4
RSET Alim_M5
RSET Alim_M6
RSET rm_transporte

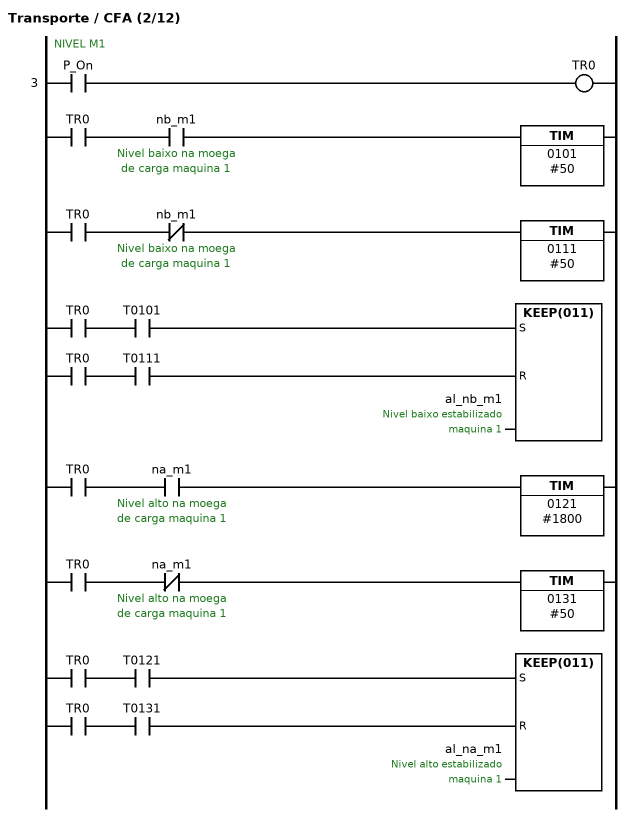
; rung 3: NIVEL M1
LD P_On
OUT TR0
AND nb_m1  ; Nivel baixo na moega de carga maquina 1
TIM 0101 #50
LD TR0
ANDNOT nb_m1  ; Nivel baixo na moega de carga maquina 1
TIM 0111 #50
LD TR0
AND T0101
LD TR0
AND T0111
KEEP(011) al_nb_m1  ; Nivel baixo estabilizado maquina 1
LD TR0
AND na_m1  ; Nivel alto na moega de carga maquina 1
TIM 0121 #1800
LD TR0
ANDNOT na_m1  ; Nivel alto na moega de carga maquina 1
TIM 0131 #50
LD TR0
AND T0121
LD TR0
AND T0131
KEEP(011) al_na_m1  ; Nivel alto estabilizado maquina 1

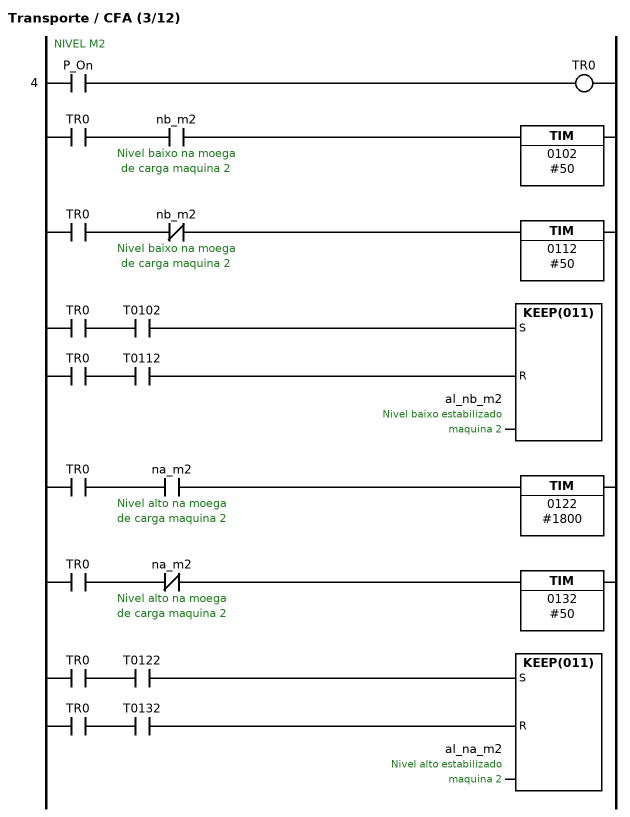
; rung 4: NIVEL M2
LD P_On
OUT TR0
AND nb_m2  ; Nivel baixo na moega de carga maquina 2
TIM 0102 #50
LD TR0
ANDNOT nb_m2  ; Nivel baixo na moega de carga maquina 2
TIM 0112 #50
LD TR0
AND T0102
LD TR0
AND T0112
KEEP(011) al_nb_m2  ; Nivel baixo estabilizado maquina 2
LD TR0
AND na_m2  ; Nivel alto na moega de carga maquina 2
TIM 0122 #1800
LD TR0
ANDNOT na_m2  ; Nivel alto na moega de carga maquina 2
TIM 0132 #50
LD TR0
AND T0122
LD TR0
AND T0132
KEEP(011) al_na_m2  ; Nivel alto estabilizado maquina 2

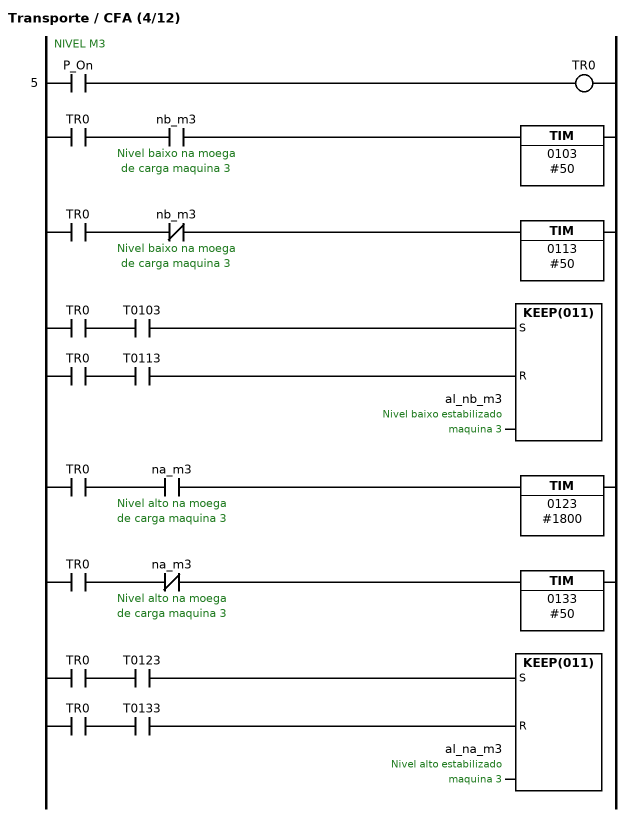
; rung 5: NIVEL M3
LD P_On
OUT TR0
AND nb_m3  ; Nivel baixo na moega de carga maquina 3
TIM 0103 #50
LD TR0
ANDNOT nb_m3  ; Nivel baixo na moega de carga maquina 3
TIM 0113 #50
LD TR0
AND T0103
LD TR0
AND T0113
KEEP(011) al_nb_m3  ; Nivel baixo estabilizado maquina 3
LD TR0
AND na_m3  ; Nivel alto na moega de carga maquina 3
TIM 0123 #1800
LD TR0
ANDNOT na_m3  ; Nivel alto na moega de carga maquina 3
TIM 0133 #50
LD TR0
AND T0123
LD TR0
AND T0133
KEEP(011) al_na_m3  ; Nivel alto estabilizado maquina 3

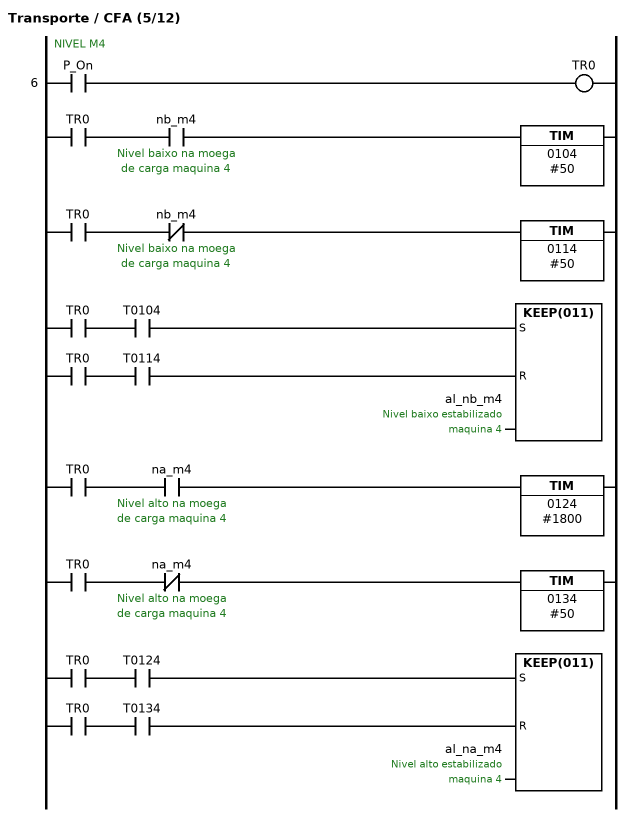
; rung 6: NIVEL M4
LD P_On
OUT TR0
AND nb_m4  ; Nivel baixo na moega de carga maquina 4
TIM 0104 #50
LD TR0
ANDNOT nb_m4  ; Nivel baixo na moega de carga maquina 4
TIM 0114 #50
LD TR0
AND T0104
LD TR0
AND T0114
KEEP(011) al_nb_m4  ; Nivel baixo estabilizado maquina 4
LD TR0
AND na_m4  ; Nivel alto na moega de carga maquina 4
TIM 0124 #1800
LD TR0
ANDNOT na_m4  ; Nivel alto na moega de carga maquina 4
TIM 0134 #50
LD TR0
AND T0124
LD TR0
AND T0134
KEEP(011) al_na_m4  ; Nivel alto estabilizado maquina 4

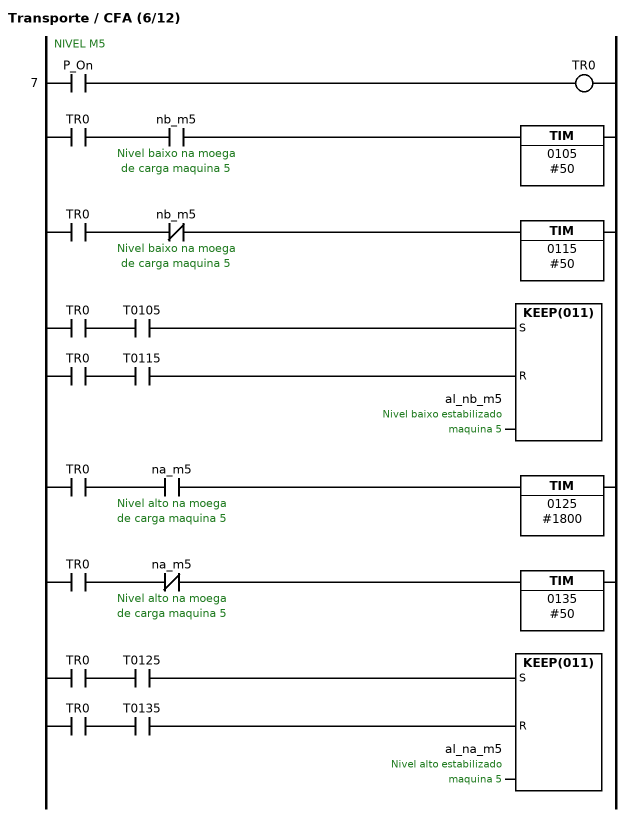
; rung 7: NIVEL M5
LD P_On
OUT TR0
AND nb_m5  ; Nivel baixo na moega de carga maquina 5
TIM 0105 #50
LD TR0
ANDNOT nb_m5  ; Nivel baixo na moega de carga maquina 5
TIM 0115 #50
LD TR0
AND T0105
LD TR0
AND T0115
KEEP(011) al_nb_m5  ; Nivel baixo estabilizado maquina 5
LD TR0
AND na_m5  ; Nivel alto na moega de carga maquina 5
TIM 0125 #1800
LD TR0
ANDNOT na_m5  ; Nivel alto na moega de carga maquina 5
TIM 0135 #50
LD TR0
AND T0125
LD TR0
AND T0135
KEEP(011) al_na_m5  ; Nivel alto estabilizado maquina 5

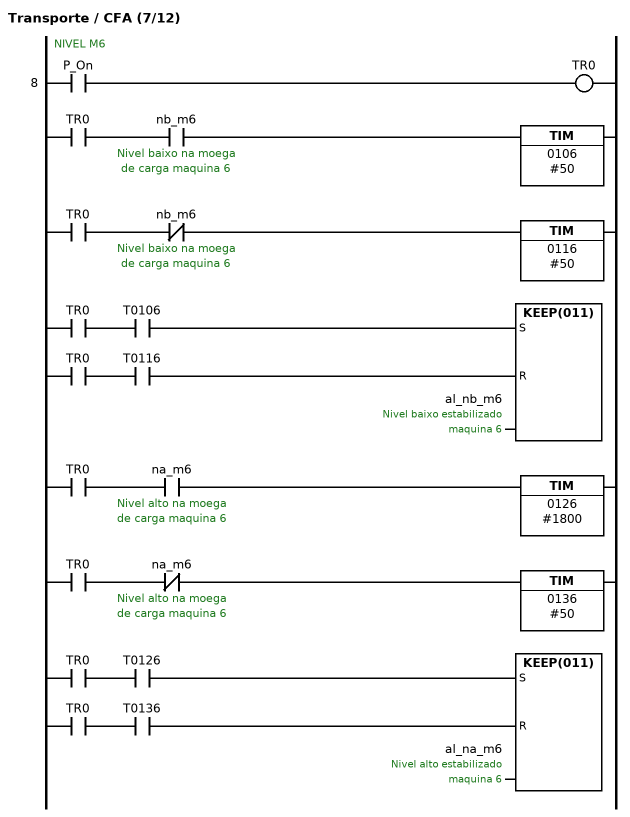
; rung 8: NIVEL M6
LD P_On
OUT TR0
AND nb_m6  ; Nivel baixo na moega de carga maquina 6
TIM 0106 #50
LD TR0
ANDNOT nb_m6  ; Nivel baixo na moega de carga maquina 6
TIM 0116 #50
LD TR0
AND T0106
LD TR0
AND T0116
KEEP(011) al_nb_m6  ; Nivel baixo estabilizado maquina 6
LD TR0
AND na_m6  ; Nivel alto na moega de carga maquina 6
TIM 0126 #1800
LD TR0
ANDNOT na_m6  ; Nivel alto na moega de carga maquina 6
TIM 0136 #50
LD TR0
AND T0126
LD TR0
AND T0136
KEEP(011) al_na_m6  ; Nivel alto estabilizado maquina 6

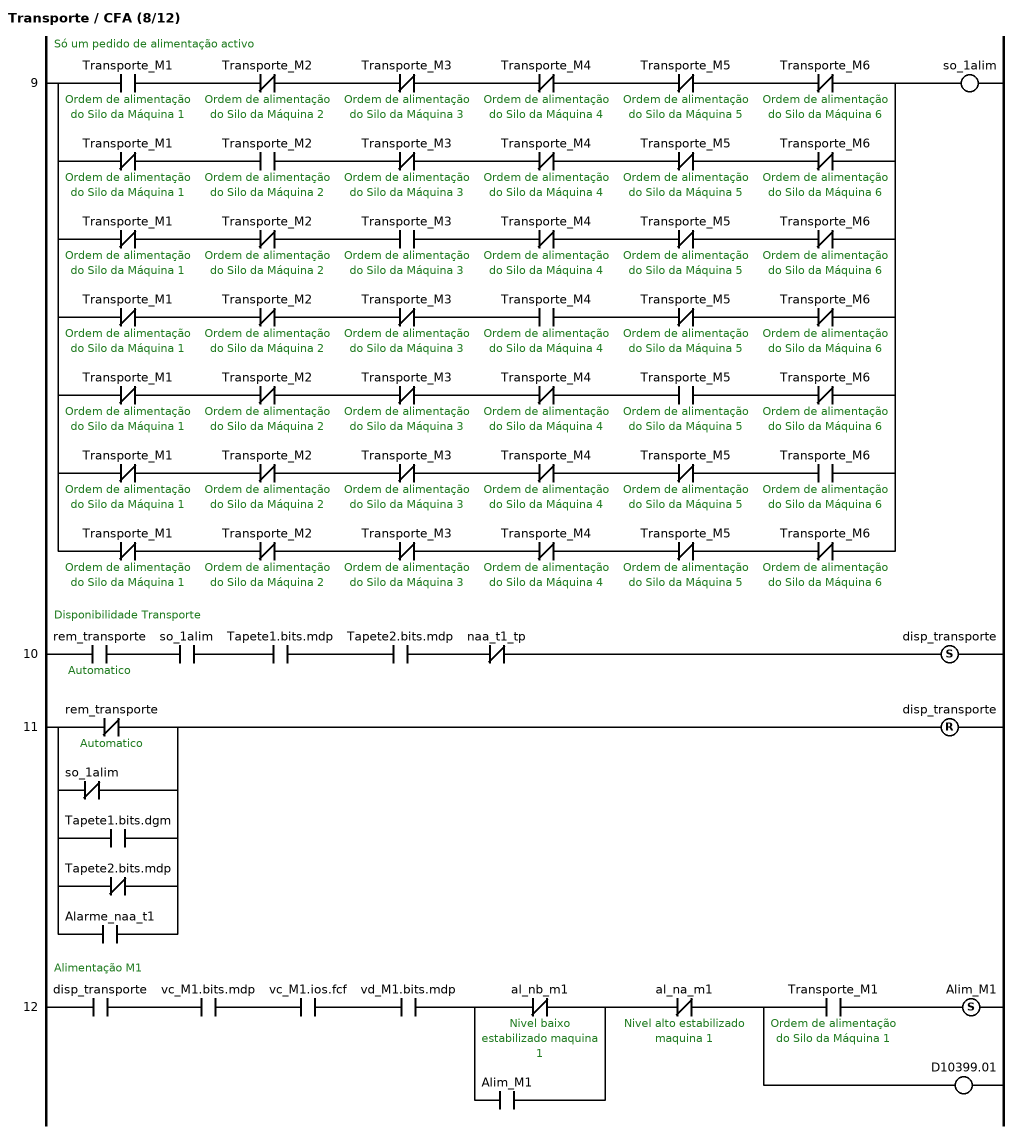
; rung 9: Só um pedido de alimentação activo
LD Transporte_M1  ; Ordem de alimentação do Silo da Máquina 1
ANDNOT Transporte_M2  ; Ordem de alimentação do Silo da Máquina 2
ANDNOT Transporte_M3  ; Ordem de alimentação do Silo da Máquina 3
ANDNOT Transporte_M4  ; Ordem de alimentação do Silo da Máquina 4
ANDNOT Transporte_M5  ; Ordem de alimentação do Silo da Máquina 5
ANDNOT Transporte_M6  ; Ordem de alimentação do Silo da Máquina 6
LDNOT Transporte_M1  ; Ordem de alimentação do Silo da Máquina 1
AND Transporte_M2  ; Ordem de alimentação do Silo da Máquina 2
ANDNOT Transporte_M3  ; Ordem de alimentação do Silo da Máquina 3
ANDNOT Transporte_M4  ; Ordem de alimentação do Silo da Máquina 4
ANDNOT Transporte_M5  ; Ordem de alimentação do Silo da Máquina 5
ANDNOT Transporte_M6  ; Ordem de alimentação do Silo da Máquina 6
ORLD
LDNOT Transporte_M1  ; Ordem de alimentação do Silo da Máquina 1
ANDNOT Transporte_M2  ; Ordem de alimentação do Silo da Máquina 2
AND Transporte_M3  ; Ordem de alimentação do Silo da Máquina 3
ANDNOT Transporte_M4  ; Ordem de alimentação do Silo da Máquina 4
ANDNOT Transporte_M5  ; Ordem de alimentação do Silo da Máquina 5
ANDNOT Transporte_M6  ; Ordem de alimentação do Silo da Máquina 6
ORLD
LDNOT Transporte_M1  ; Ordem de alimentação do Silo da Máquina 1
ANDNOT Transporte_M2  ; Ordem de alimentação do Silo da Máquina 2
ANDNOT Transporte_M3  ; Ordem de alimentação do Silo da Máquina 3
AND Transporte_M4  ; Ordem de alimentação do Silo da Máquina 4
ANDNOT Transporte_M5  ; Ordem de alimentação do Silo da Máquina 5
ANDNOT Transporte_M6  ; Ordem de alimentação do Silo da Máquina 6
ORLD
LDNOT Transporte_M1  ; Ordem de alimentação do Silo da Máquina 1
ANDNOT Transporte_M2  ; Ordem de alimentação do Silo da Máquina 2
ANDNOT Transporte_M3  ; Ordem de alimentação do Silo da Máquina 3
ANDNOT Transporte_M4  ; Ordem de alimentação do Silo da Máquina 4
AND Transporte_M5  ; Ordem de alimentação do Silo da Máquina 5
ANDNOT Transporte_M6  ; Ordem de alimentação do Silo da Máquina 6
ORLD
LDNOT Transporte_M1  ; Ordem de alimentação do Silo da Máquina 1
ANDNOT Transporte_M2  ; Ordem de alimentação do Silo da Máquina 2
ANDNOT Transporte_M3  ; Ordem de alimentação do Silo da Máquina 3
ANDNOT Transporte_M4  ; Ordem de alimentação do Silo da Máquina 4
ANDNOT Transporte_M5  ; Ordem de alimentação do Silo da Máquina 5
AND Transporte_M6  ; Ordem de alimentação do Silo da Máquina 6
ORLD
LDNOT Transporte_M1  ; Ordem de alimentação do Silo da Máquina 1
ANDNOT Transporte_M2  ; Ordem de alimentação do Silo da Máquina 2
ANDNOT Transporte_M3  ; Ordem de alimentação do Silo da Máquina 3
ANDNOT Transporte_M4  ; Ordem de alimentação do Silo da Máquina 4
ANDNOT Transporte_M5  ; Ordem de alimentação do Silo da Máquina 5
ANDNOT Transporte_M6  ; Ordem de alimentação do Silo da Máquina 6
ORLD
OUT so_1alim
; rung 10: Disponibilidade Transporte
LD rem_transporte  ; Automatico
AND so_1alim
AND Tapete1.bits.mdp
AND Tapete2.bits.mdp
ANDNOT naa_t1_tp
SET disp_transporte
; rung 11
LDNOT rem_transporte  ; Automatico
ORNOT so_1alim
OR Tapete1.bits.dgm
ORNOT Tapete2.bits.mdp
OR Alarme_naa_t1
RSET disp_transporte
; rung 12: Alimentação M1
LD disp_transporte
AND vc_M1.bits.mdp
AND vc_M1.ios.fcf
AND vd_M1.bits.mdp
LDNOT al_nb_m1  ; Nivel baixo estabilizado maquina 1
OR Alim_M1
ANDLD
ANDNOT al_na_m1  ; Nivel alto estabilizado maquina 1
OUT TR0
AND Transporte_M1  ; Ordem de alimentação do Silo da Máquina 1
SET Alim_M1
LD TR0
OUT D10399.01

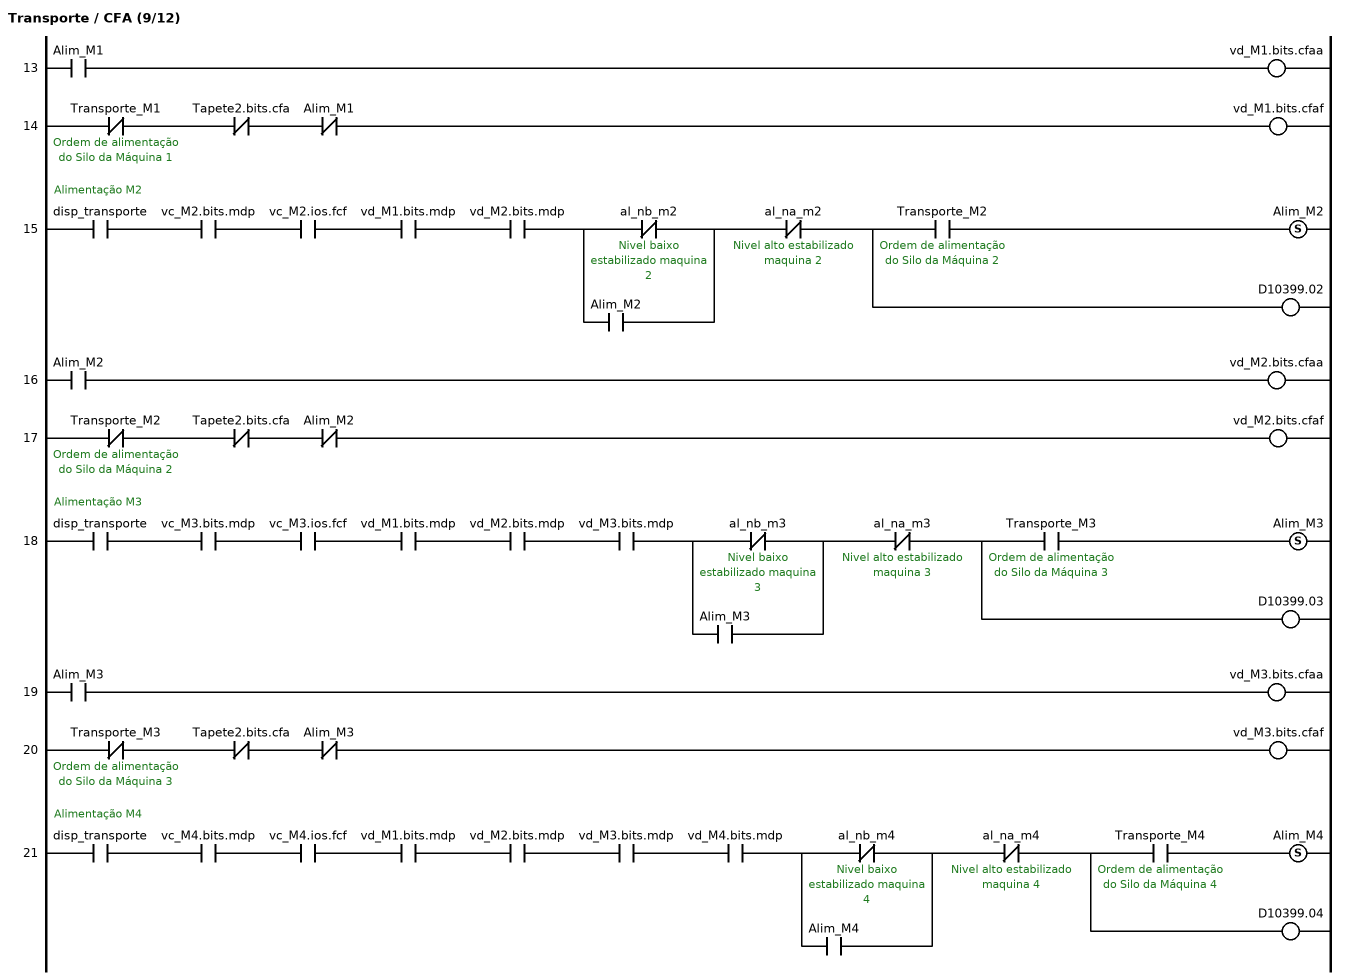
; rung 13
LD Alim_M1
OUT vd_M1.bits.cfaa
; rung 14
LDNOT Transporte_M1  ; Ordem de alimentação do Silo da Máquina 1
ANDNOT Tapete2.bits.cfa
ANDNOT Alim_M1
OUT vd_M1.bits.cfaf
; rung 15: Alimentação M2
LD disp_transporte
AND vc_M2.bits.mdp
AND vc_M2.ios.fcf
AND vd_M1.bits.mdp
AND vd_M2.bits.mdp
LDNOT al_nb_m2  ; Nivel baixo estabilizado maquina 2
OR Alim_M2
ANDLD
ANDNOT al_na_m2  ; Nivel alto estabilizado maquina 2
OUT TR0
AND Transporte_M2  ; Ordem de alimentação do Silo da Máquina 2
SET Alim_M2
LD TR0
OUT D10399.02
; rung 16
LD Alim_M2
OUT vd_M2.bits.cfaa
; rung 17
LDNOT Transporte_M2  ; Ordem de alimentação do Silo da Máquina 2
ANDNOT Tapete2.bits.cfa
ANDNOT Alim_M2
OUT vd_M2.bits.cfaf
; rung 18: Alimentação M3
LD disp_transporte
AND vc_M3.bits.mdp
AND vc_M3.ios.fcf
AND vd_M1.bits.mdp
AND vd_M2.bits.mdp
AND vd_M3.bits.mdp
LDNOT al_nb_m3  ; Nivel baixo estabilizado maquina 3
OR Alim_M3
ANDLD
ANDNOT al_na_m3  ; Nivel alto estabilizado maquina 3
OUT TR0
AND Transporte_M3  ; Ordem de alimentação do Silo da Máquina 3
SET Alim_M3
LD TR0
OUT D10399.03
; rung 19
LD Alim_M3
OUT vd_M3.bits.cfaa
; rung 20
LDNOT Transporte_M3  ; Ordem de alimentação do Silo da Máquina 3
ANDNOT Tapete2.bits.cfa
ANDNOT Alim_M3
OUT vd_M3.bits.cfaf
; rung 21: Alimentação M4
LD disp_transporte
AND vc_M4.bits.mdp
AND vc_M4.ios.fcf
AND vd_M1.bits.mdp
AND vd_M2.bits.mdp
AND vd_M3.bits.mdp
AND vd_M4.bits.mdp
LDNOT al_nb_m4  ; Nivel baixo estabilizado maquina 4
OR Alim_M4
ANDLD
ANDNOT al_na_m4  ; Nivel alto estabilizado maquina 4
OUT TR0
AND Transporte_M4  ; Ordem de alimentação do Silo da Máquina 4
SET Alim_M4
LD TR0
OUT D10399.04

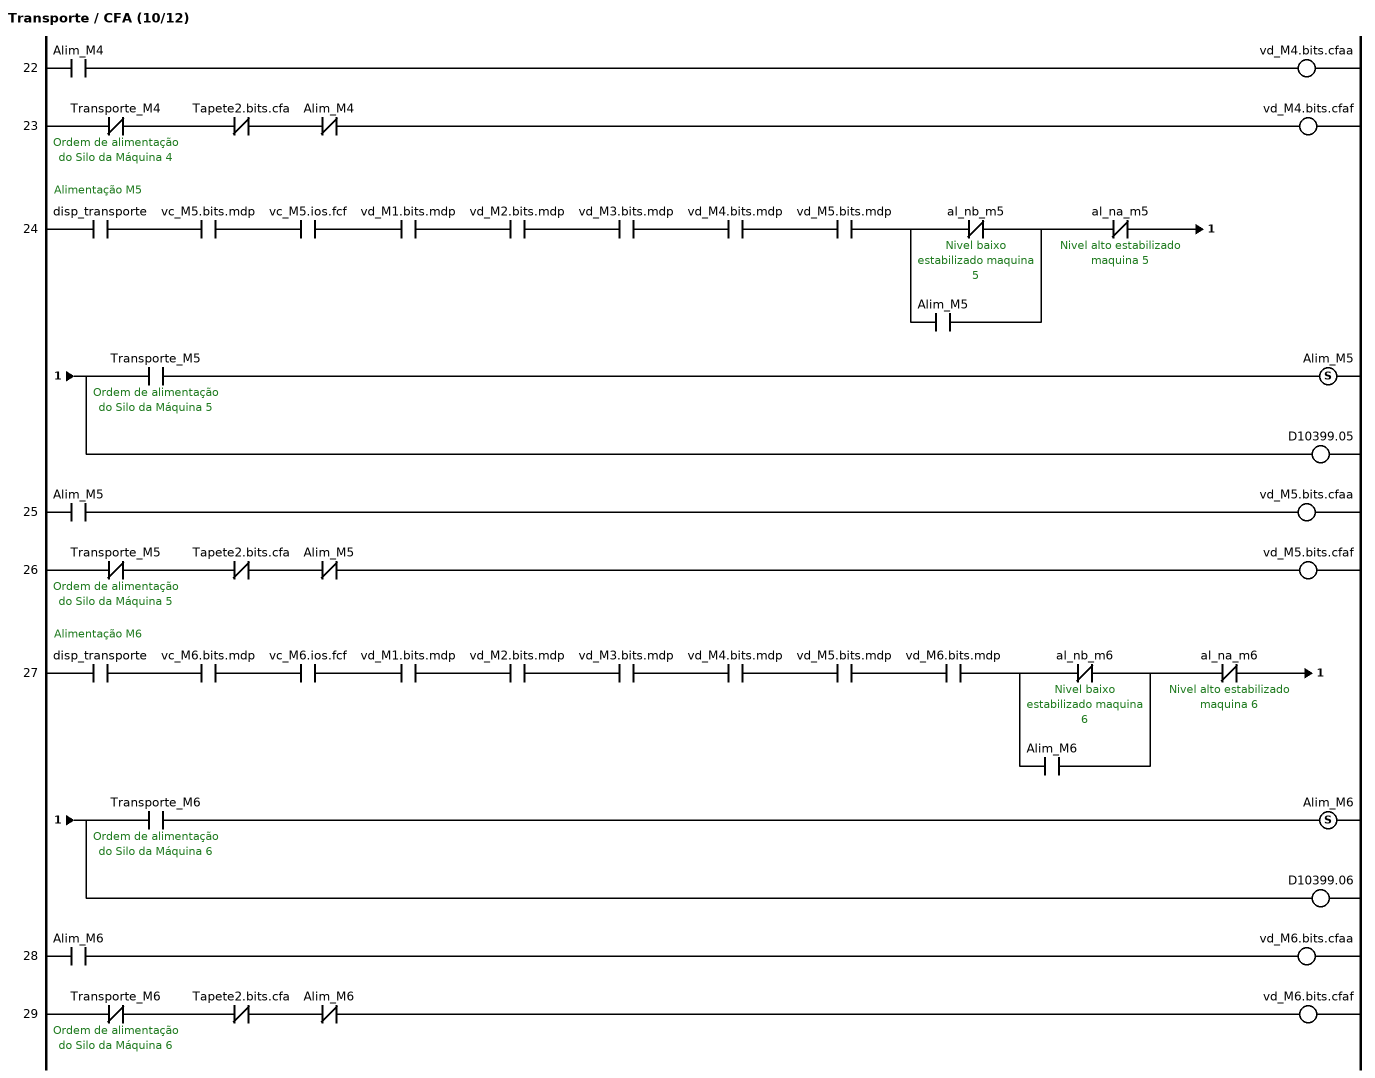
; rung 22
LD Alim_M4
OUT vd_M4.bits.cfaa
; rung 23
LDNOT Transporte_M4  ; Ordem de alimentação do Silo da Máquina 4
ANDNOT Tapete2.bits.cfa
ANDNOT Alim_M4
OUT vd_M4.bits.cfaf
; rung 24: Alimentação M5
LD disp_transporte
AND vc_M5.bits.mdp
AND vc_M5.ios.fcf
AND vd_M1.bits.mdp
AND vd_M2.bits.mdp
AND vd_M3.bits.mdp
AND vd_M4.bits.mdp
AND vd_M5.bits.mdp
LDNOT al_nb_m5  ; Nivel baixo estabilizado maquina 5
OR Alim_M5
ANDLD
ANDNOT al_na_m5  ; Nivel alto estabilizado maquina 5
OUT TR0
AND Transporte_M5  ; Ordem de alimentação do Silo da Máquina 5
SET Alim_M5
LD TR0
OUT D10399.05
; rung 25
LD Alim_M5
OUT vd_M5.bits.cfaa
; rung 26
LDNOT Transporte_M5  ; Ordem de alimentação do Silo da Máquina 5
ANDNOT Tapete2.bits.cfa
ANDNOT Alim_M5
OUT vd_M5.bits.cfaf
; rung 27: Alimentação M6
LD disp_transporte
AND vc_M6.bits.mdp
AND vc_M6.ios.fcf
AND vd_M1.bits.mdp
AND vd_M2.bits.mdp
AND vd_M3.bits.mdp
AND vd_M4.bits.mdp
AND vd_M5.bits.mdp
AND vd_M6.bits.mdp
LDNOT al_nb_m6  ; Nivel baixo estabilizado maquina 6
OR Alim_M6
ANDLD
ANDNOT al_na_m6  ; Nivel alto estabilizado maquina 6
OUT TR0
AND Transporte_M6  ; Ordem de alimentação do Silo da Máquina 6
SET Alim_M6
LD TR0
OUT D10399.06
; rung 28
LD Alim_M6
OUT vd_M6.bits.cfaa
; rung 29
LDNOT Transporte_M6  ; Ordem de alimentação do Silo da Máquina 6
ANDNOT Tapete2.bits.cfa
ANDNOT Alim_M6
OUT vd_M6.bits.cfaf

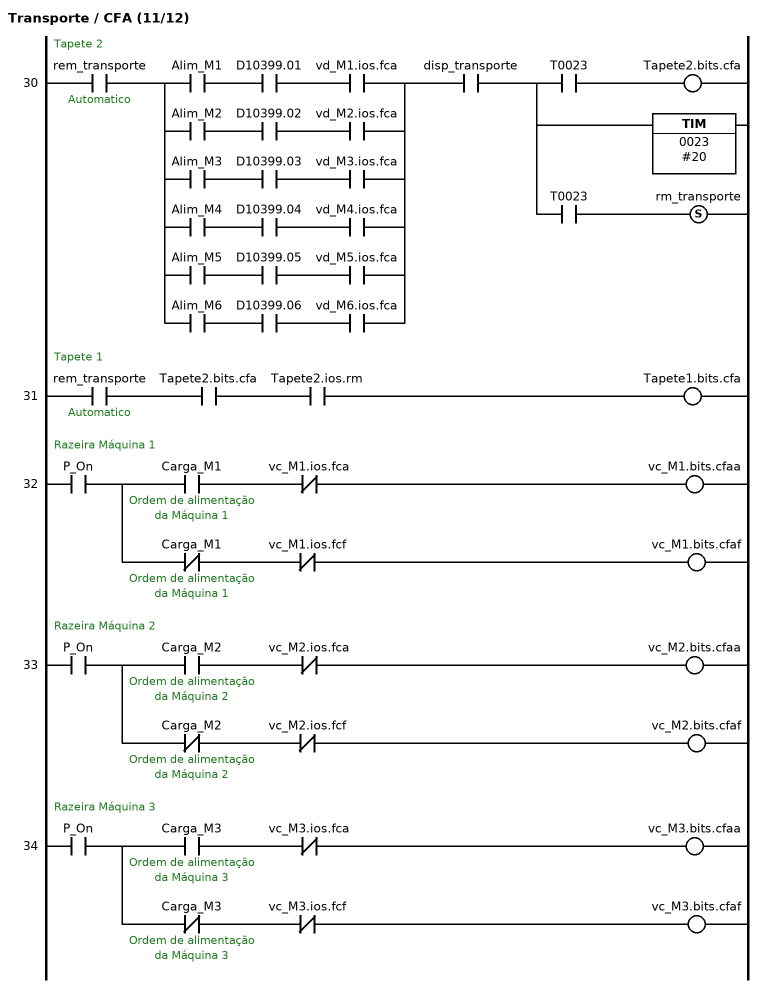
; rung 30: Tapete 2
LD rem_transporte  ; Automatico
LD Alim_M1
AND D10399.01
AND vd_M1.ios.fca
LD Alim_M2
AND D10399.02
AND vd_M2.ios.fca
ORLD
LD Alim_M3
AND D10399.03
AND vd_M3.ios.fca
ORLD
LD Alim_M4
AND D10399.04
AND vd_M4.ios.fca
ORLD
LD Alim_M5
AND D10399.05
AND vd_M5.ios.fca
ORLD
LD Alim_M6
AND D10399.06
AND vd_M6.ios.fca
ORLD
ANDLD
AND disp_transporte
OUT TR0
AND T0023
OUT Tapete2.bits.cfa
LD TR0
TIM 0023 #20
AND T0023
SET rm_transporte
; rung 31: Tapete 1
LD rem_transporte  ; Automatico
AND Tapete2.bits.cfa
AND Tapete2.ios.rm
OUT Tapete1.bits.cfa
; rung 32: Razeira Máquina 1
LD P_On
OUT TR0
AND Carga_M1  ; Ordem de alimentação da Máquina 1
ANDNOT vc_M1.ios.fca
OUT vc_M1.bits.cfaa
LD TR0
ANDNOT Carga_M1  ; Ordem de alimentação da Máquina 1
ANDNOT vc_M1.ios.fcf
OUT vc_M1.bits.cfaf
; rung 33: Razeira Máquina 2
LD P_On
OUT TR0
AND Carga_M2  ; Ordem de alimentação da Máquina 2
ANDNOT vc_M2.ios.fca
OUT vc_M2.bits.cfaa
LD TR0
ANDNOT Carga_M2  ; Ordem de alimentação da Máquina 2
ANDNOT vc_M2.ios.fcf
OUT vc_M2.bits.cfaf
; rung 34: Razeira Máquina 3
LD P_On
OUT TR0
AND Carga_M3  ; Ordem de alimentação da Máquina 3
ANDNOT vc_M3.ios.fca
OUT vc_M3.bits.cfaa
LD TR0
ANDNOT Carga_M3  ; Ordem de alimentação da Máquina 3
ANDNOT vc_M3.ios.fcf
OUT vc_M3.bits.cfaf

